(* IEC 61131-3 sources: Codesys/ddyut/src, 26 files *)

(* ---- E_PumpType.st ---- *)
(* ============================================================ *)
(* E_PumpType — тип преобразователя частоты ELHART             *)
(* ============================================================ *)
(* === ИЗМЕНЕНО === MINI удалён (в проектах его не было — была   *)
(* ошибка типа). Теперь два типа: PUMP (EMD-PUMP) и VL           *)
(* (EMD-VL/VH, векторный). Обработка обоих — в FB_Pump.          *)
(*                                                              *)
(* Тип каждого ПЧ задаётся в массиве GVL.ePumpType[1..cPumpCount] *)
(* (RETAIN). Автоопределение PUMP/VL по сигнатурному регистру —   *)
(* см. комментарий в PRG_Pumps (пока задаётся вручную).          *)
(* ============================================================ *)
TYPE E_PumpType :
(
    PUMP := 0,   // EMD-PUMP (F-коды, задание частоты в Гц ×100 → 0x2001)
    VL   := 1    // EMD-VL/VH (P-группы, задание в % → 0x1000, статус 0x3000)
);
END_TYPE

(* ---- GVL.st ---- *)
(* ============================================================ *)
(* GVL — Глобальные переменные проекта ДДЮТ                     *)
(* (на основе Fontan_V1 / Саки Пруд)                            *)
(*                                                              *)
(* ШИНА Modbus RTU / RS-485:                                   *)
(*   COM1 (Modbus_COM), 9600/8/N/1:                            *)
(*     Адрес 1  — МВ110-16Д   (16 дискретных входов DI1..DI11) *)
(*     Адрес 2  — МУ110-16Р   (16 дискретных выходов DO1..DO16)*)
(*     Аналогового модуля МВ110-8А на ДДЮТ НЕТ.                *)
(*   COM2 (Modbus_COM_2):                                       *)
(*     Адрес 41 — ELHART EMD-PUMP 1 (насос фонтана, индекс 1)  *)
(*     Адрес 42 — ELHART EMD-PUMP 2 (насос фонтана, индекс 2)  *)
(*   === ДДЮТ:ИЗМЕНЕНО === Насосы COM2 — это насосы фонтана    *)
(*   (клапаны/форсунки), НЕ фильтрационные, как было в Саки.    *)
(*   Признак работы фильтрации приходит отдельно на DI5.        *)
(* ============================================================ *)

(* ============================================================ *)
(* КОНСТАНТЫ СИСТЕМЫ                                            *)
(* ============================================================ *)
VAR_GLOBAL CONSTANT
    cPumpCount   : INT  := 2;        // количество насосов (2 × EMD-PUMP)
    cDI_Count    : INT  := 16;       // дискретных входов МВ110
    cDO_Count    : INT  := 16;       // дискретных выходов МУ110
    cMaxFreq     : REAL := 50.0;     // максимальная частота, Гц
    cMinFreq     : REAL := 0.0;      // минимальная частота, Гц
    cMinTime     : REAL := 0.1;      // мин. время разгона/торможения, с
    cMaxTime     : REAL := 6000.0;   // макс. время разгона/торможения, с
    cMaxCurrent  : REAL := 999.9;    // потолок номинального тока, А
    cMaxVoltage  : REAL := 500.0;    // потолок номинального напряжения, В
    cMaxOverheat : INT  := 150;      // потолок уровня перегрева, °C
    cMinOverheat : INT  := 40;       // минимум уровня перегрева, °C
END_VAR

(* ============================================================ *)
(* RETAIN-переменные (хранятся при отключении питания)         *)
(* ============================================================ *)
VAR_GLOBAL RETAIN
    (* Тип каждого ПЧ. Оба насоса — EMD-PUMP.                   *)
    (* ВНИМАНИЕ: изменение требует Reset cold контроллера.      *)
    ePumpType : ARRAY[1..cPumpCount] OF E_PumpType :=
        [E_PumpType.PUMP, E_PumpType.PUMP];

    (* === ДДЮТ:ИЗМЕНЕНО (round 7, ФИНАЛЬНАЯ СХЕМА) — ЖУРНАЛ ПЧ === *)
    (* Та же схема сдвига, что у журнала фонтана (см. подробный комментарий  *)
    (* в GVL_Fountain.st) — позиция 1 всегда самая свежая запись, при новой  *)
    (* записи всё сдвигается на 1 вниз, самая старая (позиция 30) выпадает.  *)
    (* Размер: 30 записей (как настроено), длина ячейки 65 (полное время     *)
    (* ДД.ММ.ГГ ЧЧ:ММ:СС + номер ПЧ + название параметра + два REAL-значения *)
    (* — уже было впритык на 65, оставлен без изменений по твоей настройке,  *)
    (* но следи, не обрезаются ли самые длинные названия типа                *)
    (* "Огр.тока.разг" — если увидишь обрыв текста, увеличь до 80-90).       *)
    aPumpLog       : ARRAY[1..30] OF WSTRING(65);
    iPumpLogCount  : INT;   // сколько записей реально заполнено (0..30)

    (* Флаг "задержка ошибки 0x02C0 уже записана в ПЧ" — RETAIN *)
    xErrDelayWritten : ARRAY[1..cPumpCount] OF BOOL := [cPumpCount(FALSE)];

    (* Флаг "параметр дисплея Fout (регистр 0) уже записан" — RETAIN *)
    xDispParamWritten : ARRAY[1..cPumpCount] OF BOOL := [cPumpCount(FALSE)];
END_VAR

(* ============================================================ *)
(* ГЛОБАЛЬНЫЕ ПЕРЕМЕННЫЕ                                        *)
(* ============================================================ *)
VAR_GLOBAL

    (* ========================================================= *)
    (* БЛОК 1: СОСТОЯНИЕ СИСТЕМЫ                                 *)
    (* ========================================================= *)
    xSystemState     : BOOL := TRUE;
    sSystemStateText : WSTRING(20);
    iErrors          : INT  := 0;
    iWorkCount       : INT  := 0;
    iStopCount       : INT  := 0;
    xAnyAlarm        : BOOL := FALSE;
    iErrorsPumps     : INT  := 0;
    iErrorsModules   : INT  := 0;
    iErrorsFountain  : INT  := 0;

    (* ========================================================= *)
    (* БЛОК 2: НАВИГАЦИЯ И ИНТЕРФЕЙС HMI                         *)
    (* ========================================================= *)
    xMenuOpen      : BOOL := TRUE;
    iCurrentScreen : INT  := 1;
    iSelPump       : INT  := 1;

    (* ========================================================= *)
    (* БЛОК 3: РЕЖИМ ОТЛАДКИ RS-485                              *)
    (* ========================================================= *)
    xDebugModeAll      : BOOL := FALSE;
    xDebugModeAll_Prev : BOOL := FALSE;

    xDebugModePump      : ARRAY[1..cPumpCount] OF BOOL := [cPumpCount(FALSE)];
    xDebugModePump_Prev : ARRAY[1..cPumpCount] OF BOOL := [cPumpCount(FALSE)];

    xApplyParamsAll  : BOOL := FALSE;
    xApplyParamsPump : ARRAY[1..cPumpCount] OF BOOL := [cPumpCount(FALSE)];

    (* ========================================================= *)
    (* ТРИГГЕРЫ ЧТЕНИЯ/ЗАПИСИ (конфигуратор-стиль)               *)
    (* ========================================================= *)
    xReadAllPump  : ARRAY[1..cPumpCount] OF BOOL := [cPumpCount(FALSE)];
    xReadAllAsk   : BOOL := FALSE;

    xWriteAllPump : ARRAY[1..cPumpCount] OF BOOL := [cPumpCount(FALSE)];
    xWriteAllAsk  : BOOL := FALSE;
    xWriteAllConfirm : BOOL := FALSE;

    xWr_AccTime      : ARRAY[1..cPumpCount] OF BOOL := [cPumpCount(FALSE)]; // 0x006B
    xWr_DecTime      : ARRAY[1..cPumpCount] OF BOOL := [cPumpCount(FALSE)]; // 0x006C
    xWr_MaxFreq      : ARRAY[1..cPumpCount] OF BOOL := [cPumpCount(FALSE)]; // 0x0069
    xWr_MinFreq      : ARRAY[1..cPumpCount] OF BOOL := [cPumpCount(FALSE)]; // 0x006A
    xWr_MotorCurrent : ARRAY[1..cPumpCount] OF BOOL := [cPumpCount(FALSE)]; // 0x00D2
    xWr_MotorVoltage : ARRAY[1..cPumpCount] OF BOOL := [cPumpCount(FALSE)]; // 0x00D1
    xWr_OverCurLevel : ARRAY[1..cPumpCount] OF BOOL := [cPumpCount(FALSE)]; // 0x01A7
    xWr_OverCurTime  : ARRAY[1..cPumpCount] OF BOOL := [cPumpCount(FALSE)]; // 0x01A8
    xWr_OverVoltProt : ARRAY[1..cPumpCount] OF BOOL := [cPumpCount(FALSE)]; // 0x019B
    xWr_Overheat     : ARRAY[1..cPumpCount] OF BOOL := [cPumpCount(FALSE)]; // 0x0325
    xWr_OverCurAcc   : ARRAY[1..cPumpCount] OF BOOL := [cPumpCount(FALSE)]; // 0x0199

    xWr_UnlockF800   : ARRAY[1..cPumpCount] OF BOOL := [cPumpCount(FALSE)]; // 0x0320
    xWr_Sources      : ARRAY[1..cPumpCount] OF BOOL := [cPumpCount(FALSE)]; // 0x0065/0x0066

    xWritePending    : ARRAY[1..cPumpCount] OF BOOL := [cPumpCount(FALSE)];
    xWaitStopForWrite : ARRAY[1..cPumpCount] OF BOOL := [cPumpCount(FALSE)];

    (* === ДДЮТ:УДАЛИТЬ ===                                       *)
    (* Раньше использовался для запроса физической остановки      *)
    (* фильтр.насоса через лампы DO6/DO8 перед записью параметров. *)
    (* На ДДЮТ ПЧ COM2 — насосы фонтана, ламп-повторов DI4/DI5     *)
    (* больше нет (DO6/DO8 свободны). Остановка перед записью      *)
    (* параметров идёт командой Modbus (см. PRG_Pumps, источник    *)
    (* RS-485) — эта переменная физически нигде не читается,      *)
    (* оставлена только для истории. Можно удалить совсем.        *)
    xReqStopFiltrForWrite : ARRAY[1..cPumpCount] OF BOOL := [cPumpCount(FALSE)];

    xFactoryResetAll  : BOOL := FALSE;
    xFactoryResetPump : ARRAY[1..cPumpCount] OF BOOL := [cPumpCount(FALSE)];

    wCmdSourceWrite  : ARRAY[1..cPumpCount] OF WORD := [cPumpCount(WORD#1)];
    wFreqSourceWrite : ARRAY[1..cPumpCount] OF WORD := [cPumpCount(WORD#3)];

    (* ========================================================= *)
    (* БЛОК 4: МВ110-16Д — ДИСКРЕТНЫЕ ВХОДЫ                      *)
    (* ========================================================= *)
    wMV110_Inputs : WORD;
    xMV110_Error  : BOOL;
    xDI           : ARRAY[1..cDI_Count] OF BOOL;
    (* === ДДЮТ:ИЗМЕНЕНО === Используются DI1..DI11.             *)
    (* Карта DI — см. PRG_Fountain блок 2.                       *)

    (* ========================================================= *)
    (* БЛОК 5: МУ110-16Р — ДИСКРЕТНЫЕ ВЫХОДЫ                     *)
    (* ========================================================= *)
    (* === ДДЮТ:ИЗМЕНЕНО === Карта DO1..DO16 — см. PRG_Fountain   *)
    (* блок 17. DO1 свет, DO2 авария, DO9 насосы, DO11 добор,     *)
    (* DO13 сухой ход/разрешение (инверсия аварии добора),        *)
    (* DO14 альгицид, DO15 биопаг, DO16 pH. Остальные свободны.   *)
    xDO                : ARRAY[1..cDO_Count] OF BOOL := [cDO_Count(FALSE)];

    wMU110_Outputs     : WORD := 0;
    wMU110_OutputsRead : WORD;
    xMU110_Error       : BOOL;

    wMU110_SafeOutputs : WORD := 0;
    xMU110_WriteSafe   : BOOL := FALSE;

    (* ========================================================= *)
    (* БЛОК 6: НАСОСЫ — ЭКЗЕМПЛЯРЫ ФУНКЦИОНАЛЬНЫХ БЛОКОВ         *)
    (* ========================================================= *)
    Pump : ARRAY[1..cPumpCount] OF FB_Pump;

    (* ========================================================= *)
    (* БЛОК 7: НАСОСЫ — ЗАДАНИЕ ОПЕРАТОРА (_Set)                 *)
    (* ========================================================= *)
    xPumpRunCmd : ARRAY[1..cPumpCount] OF BOOL := [cPumpCount(FALSE)];

    rPumpFreqSetHz          : ARRAY[1..cPumpCount] OF REAL := [cPumpCount(40.0)];
    rPumpAccTime_Set        : ARRAY[1..cPumpCount] OF REAL := [10.0, 10.0];
    rPumpDecTime_Set        : ARRAY[1..cPumpCount] OF REAL := [10.0, 10.0];
    rPumpMaxFreq_Set        : ARRAY[1..cPumpCount] OF REAL := [cPumpCount(40.0)];
    rPumpMinFreq_Set        : ARRAY[1..cPumpCount] OF REAL := [cPumpCount(0.0)];
    rPumpMotorRatedCurrent_Set : ARRAY[1..cPumpCount] OF REAL := [cPumpCount(14.9)];
    rPumpMotorRatedVoltage_Set : ARRAY[1..cPumpCount] OF REAL := [cPumpCount(380.0)];
    rPumpOverCurrentLevel_A_Set : ARRAY[1..cPumpCount] OF REAL := [cPumpCount(26.1)];
    rPumpOverCurrentTime_Set    : ARRAY[1..cPumpCount] OF REAL := [cPumpCount(5.0)];
    xPumpOverVoltProtect_Set    : ARRAY[1..cPumpCount] OF BOOL := [cPumpCount(TRUE)];
    iPumpOverheatLevel_Set      : ARRAY[1..cPumpCount] OF INT  := [cPumpCount(95)];
    iPumpOverCurAcc_Set         : ARRAY[1..cPumpCount] OF INT  := [cPumpCount(150)];

    (* ========================================================= *)
    (* БЛОК 7а: ОТЛАДКА — групповые команды и флаги окон        *)
    (* ========================================================= *)
    xDbgRunAll  : BOOL;
    xDbgStopAll : BOOL;

    xAskApply   : BOOL := FALSE;
    xAskFactory : BOOL := FALSE;
	xAskDialogStopPch : BOOL := FALSE;

    (* ========================================================= *)
    (* БЛОК 8: НАСОСЫ — ДАННЫЕ ДЛЯ ОТОБРАЖЕНИЯ НА HMI            *)
    (* ========================================================= *)
    xPumpWork      : ARRAY[1..cPumpCount] OF BOOL;
    xPumpStop      : ARRAY[1..cPumpCount] OF BOOL;
    xPumpAlarm     : ARRAY[1..cPumpCount] OF BOOL;
    xPumpReverse   : ARRAY[1..cPumpCount] OF BOOL;
    xPumpCommError : ARRAY[1..cPumpCount] OF BOOL;
    xPumpCommRaw   : ARRAY[1..cPumpCount] OF BOOL;
    tonPumpCommFilter : ARRAY[1..cPumpCount] OF TON;

    sPumpState         : ARRAY[1..cPumpCount] OF WSTRING(50);
    sPumpFaultText     : ARRAY[1..cPumpCount] OF WSTRING(100);
    sPumpTypeText      : ARRAY[1..cPumpCount] OF WSTRING(20);
    sPumpFaultLastText : ARRAY[1..cPumpCount] OF WSTRING(100);
    sPumpFault2Text    : ARRAY[1..cPumpCount] OF WSTRING(100);
    sPumpFault3Text    : ARRAY[1..cPumpCount] OF WSTRING(100);
    sPumpFault4Text    : ARRAY[1..cPumpCount] OF WSTRING(100);

    rPumpFreqSetActHz : ARRAY[1..cPumpCount] OF REAL;
    rPumpFreqActHz    : ARRAY[1..cPumpCount] OF REAL;
    rPumpCurrentActA  : ARRAY[1..cPumpCount] OF REAL;
    rPumpSpeedActRpm  : ARRAY[1..cPumpCount] OF REAL;
    rPumpDcVoltageV   : ARRAY[1..cPumpCount] OF REAL;
    iPumpTemperatureC : ARRAY[1..cPumpCount] OF INT;
    rPumpVoltageActV  : ARRAY[1..cPumpCount] OF REAL;
    rPumpRuntimeHours : ARRAY[1..cPumpCount] OF REAL;

    dwPumpLampColor : ARRAY[1..cPumpCount] OF DWORD;

    rPumpAccTime_Disp            : ARRAY[1..cPumpCount] OF REAL;
    rPumpDecTime_Disp            : ARRAY[1..cPumpCount] OF REAL;
    rPumpMaxFreq_Disp            : ARRAY[1..cPumpCount] OF REAL;
    rPumpMinFreq_Disp            : ARRAY[1..cPumpCount] OF REAL;
    rPumpMotorRatedCurrent_Disp  : ARRAY[1..cPumpCount] OF REAL;
    rPumpMotorRatedVoltage_Disp  : ARRAY[1..cPumpCount] OF REAL;
    rPumpOverCurrentLevel_A_Disp : ARRAY[1..cPumpCount] OF REAL;
    rPumpOverCurrentTime_Disp    : ARRAY[1..cPumpCount] OF REAL;
    xPumpOverVoltProtect_Disp    : ARRAY[1..cPumpCount] OF BOOL;
    sPumpOverVoltProtect : ARRAY[1..cPumpCount] OF WSTRING(20);
    iPumpOverCurrentLevel_pct_Disp : ARRAY[1..cPumpCount] OF INT;
    iPumpOverheatLevel_Disp      : ARRAY[1..cPumpCount] OF INT;
    iPumpOverCurAcc_Disp         : ARRAY[1..cPumpCount] OF INT;

    (* ========================================================= *)
    (* БЛОК 9: НАСОСЫ — ЗАПИСЬ В ПЧ (Modbus WRITE)               *)
    (* ========================================================= *)
    wPumpCmd  : ARRAY[1..cPumpCount] OF WORD;
    wPumpFreq : ARRAY[1..cPumpCount] OF WORD;

    wPumpAccTimeWrite           : ARRAY[1..cPumpCount] OF WORD;
    wPumpDecTimeWrite           : ARRAY[1..cPumpCount] OF WORD;
    wPumpMaxFreqWrite           : ARRAY[1..cPumpCount] OF WORD;
    wPumpMinFreqWrite           : ARRAY[1..cPumpCount] OF WORD;
    wPumpMotorRatedCurrentWrite : ARRAY[1..cPumpCount] OF WORD;
    wPumpMotorRatedVoltageWrite : ARRAY[1..cPumpCount] OF WORD;
    wPumpOverCurrentLevelWrite  : ARRAY[1..cPumpCount] OF WORD;
    wPumpOverCurrentTimeWrite   : ARRAY[1..cPumpCount] OF WORD;
    wPumpOverVoltProtectWrite   : ARRAY[1..cPumpCount] OF WORD;
    wPumpOverheatLevelWrite     : ARRAY[1..cPumpCount] OF WORD;
    wPumpOverCurAccWrite        : ARRAY[1..cPumpCount] OF WORD;

    wPumpDispParamWrite : ARRAY[1..cPumpCount] OF WORD := [cPumpCount(WORD#1)];

    wPumpRS_ErrDelayWrite : ARRAY[1..cPumpCount] OF WORD := [cPumpCount(WORD#5)];
    xWr_ErrDelayInit      : ARRAY[1..cPumpCount] OF BOOL := [cPumpCount(FALSE)];

    wPumpExtSettingsUnlockWrite : ARRAY[1..cPumpCount] OF WORD;
    wPumpFactoryResetWrite      : ARRAY[1..cPumpCount] OF WORD := [cPumpCount(WORD#0)];

    (* ========================================================= *)
    (* БЛОК 10: НАСОСЫ — ЧТЕНИЕ ИЗ ПЧ (Modbus READ)             *)
    (* ========================================================= *)
    wPumpFreqSetRead     : ARRAY[1..cPumpCount] OF WORD;
    wPumpFreqActual      : ARRAY[1..cPumpCount] OF WORD;
    wPumpCurrentActual   : ARRAY[1..cPumpCount] OF WORD;
    wPumpSpeedActual     : ARRAY[1..cPumpCount] OF WORD;
    wPumpDcVoltage       : ARRAY[1..cPumpCount] OF WORD;
    wPumpTemperature     : ARRAY[1..cPumpCount] OF WORD;
    wPumpPidFeedback     : ARRAY[1..cPumpCount] OF WORD;
    wPumpRuntimeHoursRaw : ARRAY[1..cPumpCount] OF WORD;
    wPumpVoltageActual   : ARRAY[1..cPumpCount] OF WORD;

    wPumpFaultLast : ARRAY[1..cPumpCount] OF WORD;
    wPumpFault2    : ARRAY[1..cPumpCount] OF WORD;
    wPumpFault3    : ARRAY[1..cPumpCount] OF WORD;
    wPumpFault4    : ARRAY[1..cPumpCount] OF WORD;

    wPumpFaultReg : ARRAY[1..cPumpCount] OF WORD;
    wPumpStatus   : ARRAY[1..cPumpCount] OF WORD;
    wPumpStopState    : ARRAY[1..cPumpCount] OF WORD;
    xPumpFullyStopped : ARRAY[1..cPumpCount] OF BOOL;

    wPumpFreqPresetRead  : ARRAY[1..cPumpCount] OF WORD;
    rPumpFreqPresetHz : ARRAY[1..cPumpCount] OF REAL;
    wPumpFreqSourceRead  : ARRAY[1..cPumpCount] OF WORD;
    wPumpCmdSourceRead   : ARRAY[1..cPumpCount] OF WORD;
    wPumpStopKeyLockRead : ARRAY[1..cPumpCount] OF WORD;
    wPumpReverseLockRead : ARRAY[1..cPumpCount] OF WORD;
    wPumpMaxFreqRead     : ARRAY[1..cPumpCount] OF WORD;
    wPumpMinFreqRead     : ARRAY[1..cPumpCount] OF WORD;
    wPumpAccTimeRaw      : ARRAY[1..cPumpCount] OF WORD;
    wPumpDecTimeRaw      : ARRAY[1..cPumpCount] OF WORD;

    wPumpStartMethodRead        : ARRAY[1..cPumpCount] OF WORD;
    wPumpStopMethodRead         : ARRAY[1..cPumpCount] OF WORD;
    wPumpStartFreqRead          : ARRAY[1..cPumpCount] OF WORD;
    wPumpStopFreqRead           : ARRAY[1..cPumpCount] OF WORD;
    wPumpMotorRatedVoltageRead  : ARRAY[1..cPumpCount] OF WORD;
    wPumpMotorRatedCurrentRead  : ARRAY[1..cPumpCount] OF WORD;
    wPumpMotorNoLoadCurrentRead : ARRAY[1..cPumpCount] OF WORD;
    wPumpMotorRatedSpeedRead    : ARRAY[1..cPumpCount] OF WORD;

    wPumpFIV_MinRead    : ARRAY[1..cPumpCount] OF WORD;
    wPumpFIV_MaxRead    : ARRAY[1..cPumpCount] OF WORD;
    wPumpFIV_FilterRead : ARRAY[1..cPumpCount] OF WORD;
    wPumpFIC_MinRead    : ARRAY[1..cPumpCount] OF WORD;
    wPumpFIC_MaxRead    : ARRAY[1..cPumpCount] OF WORD;

    wPumpFOV_MinRead : ARRAY[1..cPumpCount] OF WORD;
    wPumpFOV_MaxRead : ARRAY[1..cPumpCount] OF WORD;
    wPumpFOC_MinRead : ARRAY[1..cPumpCount] OF WORD;
    wPumpFOC_MaxRead : ARRAY[1..cPumpCount] OF WORD;

    wPumpAI_MinFreqRead  : ARRAY[1..cPumpCount] OF WORD;
    wPumpAI_MinDirRead   : ARRAY[1..cPumpCount] OF WORD;
    wPumpAI_MaxFreqRead  : ARRAY[1..cPumpCount] OF WORD;
    wPumpAI_MaxDirRead   : ARRAY[1..cPumpCount] OF WORD;
    wPumpAI_ReverseEnRead: ARRAY[1..cPumpCount] OF WORD;

    wPumpDI_FWD_Read : ARRAY[1..cPumpCount] OF WORD;
    wPumpDI_REV_Read : ARRAY[1..cPumpCount] OF WORD;
    wPumpDI_S1_Read  : ARRAY[1..cPumpCount] OF WORD;
    wPumpDI_S2_Read  : ARRAY[1..cPumpCount] OF WORD;
    wPumpDI_S3_Read  : ARRAY[1..cPumpCount] OF WORD;
    wPumpDI_S4_Read  : ARRAY[1..cPumpCount] OF WORD;
    wPumpDI_S5_Read  : ARRAY[1..cPumpCount] OF WORD;
    wPumpDI_S6_Read  : ARRAY[1..cPumpCount] OF WORD;

    wPumpDO_M01_Read   : ARRAY[1..cPumpCount] OF WORD;
    wPumpDO_M02_Read   : ARRAY[1..cPumpCount] OF WORD;
    wPumpDO_Relay_Read : ARRAY[1..cPumpCount] OF WORD;

    wPumpOverCurAccRead       : ARRAY[1..cPumpCount] OF WORD;
    wPumpOverCurSteadyRead    : ARRAY[1..cPumpCount] OF WORD;
    wPumpOverVoltProtectRead  : ARRAY[1..cPumpCount] OF WORD;
    wPumpOverCurReactionRead  : ARRAY[1..cPumpCount] OF WORD;
    wPumpOverCurrentLevelRead : ARRAY[1..cPumpCount] OF WORD;
    wPumpOverCurrentTimeRead  : ARRAY[1..cPumpCount] OF WORD;
    wPumpOverheatLevelRead    : ARRAY[1..cPumpCount] OF WORD;

    wPumpRS_BaudRead      : ARRAY[1..cPumpCount] OF WORD;
    wPumpRS_FormatRead    : ARRAY[1..cPumpCount] OF WORD;
    wPumpRS_AddrRead      : ARRAY[1..cPumpCount] OF WORD;
    wPumpRS_ErrActionRead : ARRAY[1..cPumpCount] OF WORD;
    wPumpRS_ErrDelayRead  : ARRAY[1..cPumpCount] OF WORD;

    (* ========================================================= *)
    (* БЛОК 11: VISU DEBUG — ВЫБОР НАСОСА И ДИАЛОГИ              *)
    (* ========================================================= *)
    iDebugMode         : INT;
    iDebugPumpSelected : INT := 1;
    xDlgConfirmApply   : BOOL;
    xDlgConfirmFactory : BOOL;

(* ========================================================= *)
(* БЛОК 12: ЖУРНАЛ ИЗМЕНЕНИЙ ПАРАМЕТРОВ ПЧ *)
(* ========================================================= *)
xLogClear : BOOL := FALSE;
xAskClearLog : BOOL := FALSE;

rLog_AccTime_Prev : ARRAY[1..cPumpCount] OF REAL;
rLog_DecTime_Prev : ARRAY[1..cPumpCount] OF REAL;
rLog_MaxFreq_Prev : ARRAY[1..cPumpCount] OF REAL;
rLog_MinFreq_Prev : ARRAY[1..cPumpCount] OF REAL;
rLog_MotorCur_Prev : ARRAY[1..cPumpCount] OF REAL;
rLog_MotorVolt_Prev : ARRAY[1..cPumpCount] OF REAL;
rLog_OCLevel_Prev : ARRAY[1..cPumpCount] OF REAL;
rLog_OCTime_Prev : ARRAY[1..cPumpCount] OF REAL;
xLog_OVProt_Prev : ARRAY[1..cPumpCount] OF BOOL;
iLog_Overheat_Prev : ARRAY[1..cPumpCount] OF INT;
iLog_OCAcc_Prev : ARRAY[1..cPumpCount] OF INT;
xLog_Initialized : ARRAY[1..cPumpCount] OF BOOL := [cPumpCount(FALSE)];
rtrigReadAll_Prev : ARRAY[1..cPumpCount] OF BOOL := [cPumpCount(FALSE)];

xWr_DispParam : ARRAY[1..cPumpCount] OF BOOL := [cPumpCount(FALSE)];
END_VAR

(* ---- GVL_Fountain.st ---- *)
(* ============================================================ *)
(* GVL_Fountain — переменные автоматики фонтана ДДЮТ            *)
(* (на основе Fontan_V1 / Саки Пруд)                            *)
(*                                                              *)
(* === ГЛАВНЫЕ ОТЛИЧИЯ ОТ САКИ ===                              *)
(*  - Уровень чаши: ДВА дискретных входа (DI7 нижний, DI8       *)
(*    верхний) вместо аналогового 4-20мА. Нет ямы слива.        *)
(*  - Сухой ход — отдельный вход DI6, не расчёт по см.          *)
(*  - Фильтрация: контактор фильтр.насоса на DI5 отдельно от    *)
(*    насосов COM2 (те теперь качают фонтан, не фильтруют).     *)
(*  - Нет ПР200 и резерва полива СПК (файлы сохранены, не       *)
(*    вызываются — легко вернуть).                              *)
(*  - Расчёт заката — новый (NOAA, FB_SunsetRelay), не завязан   *)
(*    ни на один DI.                                            *)
(*                                                              *)
(* КАРТА ВЫХОДОВ DO (МУ110-16Р, COM1, адрес 2):                 *)
(*   DO1  — СВЕТ                                                *)
(*   DO2  — ЛАМПА АВАРИИ (мигает)                                *)
(*   DO3..DO8, DO10, DO12 — свободны (FALSE)                    *)
(*   DO9  — НАСОСЫ ФОНТАНА                                      *)
(*   DO11 — КЛАПАН ДОБОРА (заслонка)                            *)
(*   DO13 — "сухой ход/разрешение": 1=норма, 0=авария добора    *)
(*          (после исчерпания попыток), см. PRG_Fountain блок 7 *)
(*   DO14 — АЛЬГИЦИД                                             *)
(*   DO15 — БИОПАГ / ОБЕЗЗАРАЖИВАТЕЛЬ                            *)
(*   DO16 — pH                                                  *)
(*                                                              *)
(* КАРТА ВХОДОВ DI (МВ110-16Д, COM1, адрес 1):                  *)
(*   DI1  — ПЧ1 насос фонтана (работа)                          *)
(*   DI2  — ПЧ2 насос фонтана (работа)                          *)
(*   DI3  — разрешение работы частотников                       *)
(*   DI4  — контактор УФ (мониторинг, выхода на УФ нет)         *)
(*   DI5  — контактор фильтр.насоса (наработка НФ)               *)
(*   DI6  — реле СУХОГО ХОДА (1 = вода есть)                    *)
(*   DI7  — УРОВЕНЬ 1 нижний  (0 = нужен добор)                 *)
(*   DI8  — УРОВЕНЬ 2 верхний (1 = стоп добора)                 *)
(*   DI9  — подтверждение работы pH                             *)
(*   DI10 — подтверждение работы биопаг                         *)
(*   DI11 — подтверждение работы альгицид                       *)
(*   DI12..DI16 — свободны                                       *)
(* ============================================================ *)

VAR_GLOBAL CONSTANT
    (* === ДДЮТ:УДАЛИТЬ — шкала уровня чаши по AI1 не нужна === *)
    (* Уровень чаши теперь дискретный (DI7/DI8), нет 4-20мА.     *)
    (*
    cWaterRawMin : REAL := 4.0;
    cWaterRawMax : REAL := 20.0;
    cWaterCmMin  : REAL := 0.0;
    cWaterCmMax  : REAL := 100.0;
    *)

    (* === ДДЮТ: ОСТАВЛЕНО АКТИВНЫМ === Используется только      *)
    (* файлом PRG_PolivSPK.st (сохранён, не вызывается на ДДЮТ,  *)
    (* т.к. нет ямы слива). Оставлено, чтобы файл не переставал   *)
    (* компилироваться. Если PRG_PolivSPK.st будет физически      *)
    (* удалён из проекта — эти константы тоже можно убрать.       *)
    cSlivRawMin : REAL := 4.0;
    cSlivRawMax : REAL := 20.0;
    cSlivCmMin  : REAL := 0.0;
    cSlivCmMax  : REAL := 100.0;
END_VAR

VAR_GLOBAL RETAIN
    (* === ДДЮТ:ИЗМЕНЕНО (round 7, ФИНАЛЬНАЯ СХЕМА) — ЖУРНАЛ ИЗМЕНЕНИЙ       *)
    (* ПАРАМЕТРОВ ФОНТАНА ===                                                 *)
    (* Причина, почему это массив, а не одна строка — см. round 6: WCONCAT в *)
    (* CODESYS официально ограничен 255 символами возврата, независимо от     *)
    (* объявленного размера WSTRING (https://content.helpme-codesys.com/en/  *)
    (* CODESYS String Libraries/_strlib_start_page.html).                    *)
    (* === ДДЮТ:ИЗМЕНЕНО (round 7) === СХЕМА СДВИГА (новое): позиция 1 —      *)
    (* ВСЕГДА самая последняя запись. При каждой новой записи всё, что было,  *)
    (* сдвигается на 1 позицию вниз (2→3, 1→2), новая запись садится на       *)
    (* позицию 1. Когда достигнут предел (60) — самая старая запись           *)
    (* (позиция 60) при сдвиге просто "выпадает" из массива. Это устраняет    *)
    (* необходимость в НА ЭКРАНЕ вычисляемых индексах вида                    *)
    (* "aFountainLog[iFountainLogCount-k]" — ИМЕННО такие вычисляемые         *)
    (* индексы, судя по всему, и давали "путаницу переменных" (при           *)
    (* iFountainLogCount меньше, чем число видимых на экране строк, индекс    *)
    (* уходил в 0 или отрицательное число — обращение к несуществующему       *)
    (* элементу массива в CODESYS не ошибка компиляции, а чтение "что         *)
    (* попало" из соседней памяти). Теперь на экране — ВСЕГДА статичные       *)
    (* константы 1, 2, 3... — вне диапазона массива уйти невозможно.          *)
    (* Размер: 60 записей, длина ячейки 60 символов (по прямому запросу).    *)
    (* ⚠️ С полными названиями + единицы измерения у обоих значений + пробелы*)
    (* вокруг стрелки — для записей с REAL (доза/расход, REAL_TO_WSTRING     *)
    (* может дать много знаков после запятой) возможна обрезка в конце       *)
    (* строки при длинных значениях. Если увидишь обрыв текста — увеличивай.*)
    aFountainLog       : ARRAY[1..60] OF WSTRING(60);
    iFountainLogCount  : INT;   // сколько записей реально заполнено (0..60)

    (* === ДДЮТ:НОВОЕ === Единый пароль для очистки ОБОИХ журналов        *)
    (* (ПЧ и фонтана) — числовой, проверяется в ST-коде через встроенный   *)
    (* элемент OwenVisu LoginOnlyPassWithKeysOwen. RETAIN — не теряется    *)
    (* при пропадании питания. Поменяй значение под себя (это заводское    *)
    (* значение-пример, не оставляй в эксплуатации).                       *)
    iAdminPassCorrect : INT := 1234;

    (* ===== ГЛАВНЫЕ ТУМБЛЕРЫ С ЭКРАНА ====================== *)
    xVseSist : BOOL := TRUE;
    (* === ДДЮТ:ИЗМЕНЕНО (единый селектор режимов) ===          *)
    (* Вместо двух раздельных элементов (тумблер разрешения +    *)
    (* отдельная кнопка ручного пуска) — один 3-позиционный      *)
    (* выбор на экране, который сам раскладывается на пару       *)
    (* (Enable, ManualForce). Раскладка — в PRG_Fountain.st,      *)
    (* блок 2а. Значения:                                        *)
    (*   0 = Ручной пуск (принудительно вкл, минуя автоматику)   *)
    (*   1 = Выкл (запрет) — значение по умолчанию для ЛЮБОГО     *)
    (*       некорректного индекса тоже трактуется как "выкл"    *)
    (*   2 = Авто (штатная логика с учётом всех условий)         *)
    iPumpSelect : INT := 2;   // насосы фонтана: 0=ручной,1=выкл,2=авто
    xNfEnable : BOOL := TRUE;

    (* ===== === ДДЮТ:УДАЛИТЬ — УСТАВКИ УРОВНЯ В СМ (AI1) ===== *)
    (* Уровень теперь дискретный, пороги в см не нужны.          *)
    (*
    rLevelOverflow   : REAL := 94.0;
    rLevelNorm       : REAL := 92.5;
    rLevelRefill     : REAL := 91.5;
    rLevelEmergency1 : REAL := 88.0;
    rLevelEmergency2 : REAL := 60.0;
    sLevelOverflow : WSTRING := "Уровень Перелив";
    sLevelNorm : WSTRING := "Уровень Норма";
    sLevelRefill : WSTRING := "Уровень Подпитка";
    sLevelEmergency1 : WSTRING := "Уровень Аварийный 1";
    sLevelEmergency2 : WSTRING := "Уровень Перелив Аварийный 2";
    *)

    (* ===== === ДДЮТ:ИЗМЕНЕНО — УРОВЕНЬ, КОНФИГУРИРУЕМЫЙ 2 ИЛИ 3   *)
    (* ДАТЧИКА (с экрана, кнопками/тумблером) ================= *)
    (* iLevelSensorCountPending = 2: датчики Уровень1 (DI7) и Уровень2*)
    (* (DI8).                                                        *)
    (*   Уровень1=0 (подтверждено) → СУХОЙ ХОД (запрет всего).     *)
    (*   Уровень1=1 И Уровень2=0 (подтверждено) → СТАРТ добора.    *)
    (*   Уровень2=1 (подтверждено) → "хватит", ПОСЛЕ доп.задержки  *)
    (*   iRefillOffDelayMin/Sec — СТОП добора.                     *)
    (* iLevelSensorCountPending = 3: датчики Уровень1 (DI7), Уровень2*)
    (* (DI8), Уровень3 (DI12).                                      *)
    (*   Уровень1=0 (подтверждено) → СУХОЙ ХОД (запрет всего) —     *)
    (*   РОЛЬ ТА ЖЕ, что и в режиме на 2 датчика.                   *)
    (*   Уровень2=0 (подтверждено) → СТАРТ добора (та же роль,      *)
    (*   что у Уровня2 в режиме на 2 датчика).                      *)
    (*   Уровень3=1 (подтверждено) → "хватит", ПОСЛЕ доп.задержки   *)
    (*   — СТОП добора (роль, которую в 2-датчиковом режиме играет  *)
    (*   сам Уровень2).                                             *)
    (* Итог: Уровень1 везде = сухой ход. Уровень2 везде = старт      *)
    (* добора. Разница только в том, ОТКУДА берётся сигнал "хватит":*)
    (* в 2-датчиковом режиме — снова Уровень2 (=1), в 3-датчиковом  *)
    (* — отдельный Уровень3.                                        *)
    (* === ДДЮТ:ИЗМЕНЕНО === Раньше было две переменные (Pending +   *)
    (* подтверждённая, с диалогом PIN-подтверждения в коде). Убрано  *)
    (* по твоей просьбе — защита от случайной записи теперь делается *)
    (* штатными средствами CODESYS (права доступа/пароль на элемент  *)
    (* визуализации при записи переменной), отдельная ST-логика для  *)
    (* этого не нужна. Осталась ОДНА переменная, пишется с экрана     *)
    (* напрямую, используется везде по коду как есть.                *)
    iLevelSensorCountPending : INT := 2;   // 2 или 3, пишется с экрана напрямую

    (* === ДДЮТ:УДАЛИТЬ === "потолок времени" был временной заменой   *)
    (* системы попыток (см. tRefillDurHours/tBetweenRefillHours/       *)
    (* iRefillAttemptsMax выше) — вернул как было в Саки, эта одиночная*)
    (* уставка больше не нужна.                                        *)
    (*
    iRefillMaxDurationMin : INT := 90;
    *)

    (* Гистерезис (антидребезг) КАЖДОГО датчика — свой, все         *)
    (* редактируются с экрана. По умолчанию 20 сек.                 *)
    tLevel1DebounceSec : INT := 20;  // Уровень1 (сухой ход)
    tLevel2DebounceSec : INT := 20;  // Уровень2 (старт добора; и стоп в режиме 2 датчика)
    tLevel3DebounceSec : INT := 20;  // Уровень3 (стоп добора, ТОЛЬКО режим 3 датчика)

    (* Доп. задержка ВЫКЛЮЧЕНИЯ добора после того, как "хватит"      *)
    (* подтверждено гистерезисом — чтобы не дёргать клапан сразу.   *)
    (* Задаётся в минутах+секундах с экрана. По умолчанию 2 мин 0с. *)
    (* Если поставить 0:00 — выключение происходит сразу (без доп.  *)
    (* выдержки), работает в обоих режимах (2 и 3 датчика) одинаково.*)
    iRefillOffDelayMin : INT := 2;
    iRefillOffDelaySec : INT := 0;

    (* === ДДЮТ:УДАЛИТЬ — ПАРАМЕТРЫ ЗАСЛОНКИ ПО КОНЦЕВИКАМ =========*)
    (* Не применимы — на ДДЮТ у заслонки нет концевиков/реле         *)
    (* направления, только команда клапана.                         *)
    (*
    tDamperTimeoutSec   : INT := 60;
    tOverflowDelaySec   : INT := 60;
    tLevelBlockDelaySec : INT := 10;
    tDamperConfirmSec : INT := 20;
    *)

    (* Смещение часового пояса от UTC, сек. Крым/МСК = +3ч=10800.*)
    iTimeZoneOffsetSec : INT := 10800;
    iUvNfMinRunMin : INT := 20;   // мин. непрерывной работы НФ для включения УФ, мин (перепроверить)

    (* === ДДЮТ:ВОЗВРАЩЕНО — СИСТЕМА ПОПЫТОК ДОБОРА === *)
    (* Была помечена "устарела" и заменена простым потолком времени  *)
    (* (xRefillMaxDurationAlarm) — но это было неверно: одна неудачная *)
    (* попытка (например, временно нет воды в городском водопроводе) *)
    (* не должна сразу давать аварию. Возвращена логика из Саки:      *)
    (* пробуем добраться tRefillDurHours; если не вышло — пауза       *)
    (* tBetweenRefillHours, новая попытка; после iRefillAttemptsMax   *)
    (* неудачных попыток подряд — авария, до ручного сброса.          *)
    (* xRefillMaxDurationAlarm/iRefillMaxDurationMin — УДАЛЕНЫ,       *)
    (* эта система их полностью заменяет.                             *)
    tRefillDurHours     : INT := 2;   // время на одну попытку добора, часы
    tBetweenRefillHours : INT := 12;  // пауза между неудачными попытками, часы
    iRefillAttemptsMax  : INT := 5;   // макс. число неудачных попыток подряд

    (* === ДДЮТ:УДАЛИТЬ — пороги сливного бака (нет ямы слива) === *)
    (*
    rSlivPolivOnCm : REAL := 5.0;
    rSlivDoborOnCm : REAL := 20.0;
    rSlivNormaPolivCm : REAL := 30.0;
    *)

    (* ===== ДОЗАЦИЯ pH — ТОЛЬКО РАЗРЕШЕНИЕ (без таймера) ==== *)
    (* === ДДЮТ:ИЗМЕНЕНО (единый селектор) — см. пояснение у   *)
    (* iPumpSelect выше. Раскладка в PRG_Fountain.st блок 2а.   *)
    iPhSelect : INT := 2;   // pH: 0=ручной,1=выкл,2=авто

    (* ===== ДОЗАЦИЯ АЛЬГИЦИД — === ДДЮТ:ИЗМЕНЕНО (round 3), реальные значения === *)
    iAlgSelect        : INT := 2;   // альгицид: 0=ручной,1=выкл,2=авто
    rAlgDoseMlPerDay  : REAL := 66.0;     // суточная доза, мл (ДДЮТ)
    rAlgFlowMlPerHour : REAL := 1125.0;   // расход насоса, мл/ч (ДДЮТ)

    (* ===== ДОЗАЦИЯ БИОПАГА — === ДДЮТ:ИЗМЕНЕНО (round 3), реальные значения === *)
    (* ВНИМАНИЕ — МОЯ ИНТЕРПРЕТАЦИЯ ЧИСЕЛ, ПРОВЕРЬ:                *)
    (* Ты написал расход "1.125 и 1.154" без единиц. Для альгицида *)
    (* уже подтверждено 1125 мл/ч (совпадает с "1.125" при чтении   *)
    (* точки как разделителя тысяч). По той же логике "1.154"       *)
    (* прочитано как 1154 мл/ч (а не буквально 1.154 мл/ч — при     *)
    (* таком мизерном расходе доза 33 мл выдавалась бы ~29 часов,    *)
    (* что маловероятно). Если я неправильно понял и расход         *)
    (* биопага ДЕЙСТВИТЕЛЬНО 1.154 мл/ч (не 1154) — поменяй ниже.   *)
    iBioSelect        : INT := 2;   // биопаг: 0=ручной,1=выкл,2=авто
    rBioDoseMlPerDay  : REAL := 33.0;     // суточная доза, мл (ДДЮТ)
    rBioFlowMlPerHour : REAL := 1154.0;   // расход насоса, мл/ч (ДДЮТ) — СВЕРИТЬ, см. выше

    (* ===== ОКНО ИСПРАВНОСТИ ФИЛЬТРАЦИИ ==================== *)
    iFilterMinRunMin   : INT := 30;    // порог наработки НФ, мин (перепроверить)
    iFilterWindowHours : INT := 12;    // (устар., не используется)
    iNfHealthyWindowMin : INT := 0;

    (* === ДДЮТ:НОВОЕ — счётчик промывок НФ (двухстадийный алгоритм,   *)
    (* см. блок 4а PRG_Fountain.st). RETAIN — переживает пропадание     *)
    (* питания, как и остальные счётчики/журналы в проекте.             *)
    iNfLastOnHour  : INT;   // время последнего включения НФ
    iNfLastOnMin   : INT;
    iNfLastOnDay   : INT;
    iNfLastOnMonth : INT;
    iNfLastOnYear  : INT;
    iNfFlushStage  : INT;   // 0=ждём часть 1, 1=часть 1 выполнена, ждём часть 2
    xNfFlushReady  : BOOL := TRUE;  // защита от многократного счёта подряд
    iNfFlushCount  : INT;   // счётчик завершённых промывок (обе части)
    iNfFlushHour   : INT;   // время последней завершённой промывки
    iNfFlushMin    : INT;
    iNfFlushDay    : INT;
    iNfFlushMonth  : INT;
    iNfFlushYear   : INT;

    iNfRunMinAccum    : INT;
    iNfRunSecAccum    : DINT;
    iNfHealthySecLeft : DINT;    // (устар., не исп.)
    iNfHealthyHoursLeft : INT;   // (устар., не исп.)
    iNfHealthyMinLeft   : INT;   // (устар., не исп.)
    xNfProven         : BOOL;    // (устар., не исп.)
    xNfWorkPrev       : BOOL;    // === ДДЮТ:РЕАКТИВИРОВАНО === детект фронта для счётчика промывок (было "не исп.")
    iNfContinuousRunHour : INT;
    iNfContinuousRunMin  : INT;
    iNfContinuousRunSec  : INT;

    (* === ДДЮТ:НОВОЕ — счётчик промывок НФ (двухстадийный алгоритм) === *)
    xNfFirstScanDone : BOOL;   // защита от ложного фронта на первом скане
    iNfJustEndedSec  : INT;    // длительность только что завершённого интервала работы НФ, сек

    (* ===== БЛОКИРОВКА ДОЗАЦИИ ПРИ РУЧНОЙ ФИЛЬТРАЦИИ ======== *)
    xZapretDozacii : BOOL := TRUE;

    (* ===== ЗАПРЕТ ДОБОРА ВОДЫ ФОНТАНА (с экрана) ========== *)
    (* === ДДЮТ:НОВОЕ === Единый селектор заслонки, тот же          *)
    (* паттерн (0/1/2), что у остальных узлов. Раскладка —          *)
    (* PRG_Fountain.st блок 2а: 0=Ручной → xDamperForceOpen:=TRUE    *)
    (* (открыто несмотря ни на что); 1=Выкл → xDamperForceClose:=    *)
    (* TRUE И xDamperZapretDobor:=TRUE (закрыта и запрет на новый     *)
    (* добор); 2=Авто → обе форс-переменные и запрет сняты, работает *)
    (* обычная автоматика по датчикам (гистерезис + попытки).        *)
    (* xDamperZapretDobor САМА теперь НЕ RETAIN (см. ниже, non-retain*)
    (* блок) — вычисляется из iDamperSelect, а не пишется напрямую. *)
    iDamperSelect : INT := 2;   // заслонка: 0=ручной,1=выкл,2=авто

    (* ===== СВЕТ ==================================== *)
    (* === ДДЮТ:ИЗМЕНЕНО (единый селектор, заменяет iLightMode) === *)
    (* Старое трёхрежимное iLightMode (0=ручной вкл/выкл через     *)
    (* xLightManualOn, 1=принудительно вкл, 2=по закату) упразднено*)
    (* — раскладывается в тот же паттерн (Enable, ManualForce),    *)
    (* что и у остальных узлов. "Ручной пуск" здесь = force-вкл    *)
    (* независимо от расписания (использует уже существующий      *)
    (* xLightForceOn), "Авто" = штатная работа по закату.          *)
    iLightSelect : INT  := 2;       // свет: 0=ручной,1=выкл,2=авто(закат)
    iSoundMode   : INT  := 2;       // FUTURE_SOUND
    xSoundEnable : BOOL := TRUE;    // FUTURE_SOUND

    (* ===== === ДДЮТ:ИЗМЕНЕНО (v2) — РАСЧЁТ ЗАКАТА (NOAA+рефракция) *)
    (* Координаты объекта ДДЮТ — ПОДТВЕРЖДЕНО (44.61581/33.52276). *)
    (* Формат — десятичные градусы (не град/мин/сек), как и была     *)
    (* организована переменная изначально — уточнять формат не       *)
    (* потребовалось, только сами значения.                          *)
    rSunLatitude          : REAL := 44.61581;  // широта объекта, град (-90..90)
    rSunLongitude         : REAL := 33.52276;  // долгота объекта, град (-180..180)
    (* === ДДЮТ:НОВОЕ === Запоминает долготу, на которую УЖЕ           *)
    (* среагировал автоподбор часового пояса (см. PRG_Fountain.st,     *)
    (* блок 11). По умолчанию совпадает с rSunLongitude — чтобы на     *)
    (* первом холодном старте НЕ переписать корректный дефолт          *)
    (* iChoseTimeZone=14 (+3, Москва) на неверный (см. пояснение там). *)
    rSunLongitudePrev     : REAL := 33.52276;
    (* === ДДЮТ:ИЗМЕНЕНО === часовой пояс теперь выбирается         *)
    (* КОМБОБОКСОМ через FB_TimeZoneSelect (индекс 0-23 → смещение  *)
    (* -11..+12). iChoseTimeZone — то, что крутит оператор на       *)
    (* экране ("Текстовый список", см. FB_TimeZoneSelect.st для     *)
    (* полного списка городов). 14 = Москва/Крым (+3) по умолчанию. *)
    (* === ДДЮТ:НОВОЕ === ТАКЖЕ теперь автоматически подбирается    *)
    (* ОДИН РАЗ при каждом реальном изменении долготы (не при        *)
    (* каждом цикле!) — см. PRG_Fountain.st блок 11. Если после      *)
    (* автоподбора оператор вручную поправит значение — это          *)
    (* сохранится и не будет затёрто повторно, пока долгота снова     *)
    (* не изменится.                                                  *)
    iChoseTimeZone        : INT  := 14;     // индекс часового пояса, с экрана (0..23)

    (* === ДДЮТ:ИЗМЕНЕНО (по макету экрана) === Коррекция теперь    *)
    (* ОДНО знаковое поле "+00мин"/"-00мин", а не два раздельных     *)
    (* элемента (было: минуты + отдельный тумблер раньше/позже).    *)
    (* Раскладывается на пару (iSunsetCorrectMin, xSunsetCorrectEarlier)*)
    (* — те, что реально идут на вход FB_SunsetRelay — в             *)
    (* PRG_Fountain.st блок 11, тем же приёмом, что и 3-позиционные  *)
    (* селекторы в блоке 2а.                                        *)
    iSunsetCorrectSigned  : INT  := 0;      // коррекция заката, мин, ЗНАКОВАЯ (- раньше, + позже)

    (* === ДДЮТ:ИЗМЕНЕНО === время отключения теперь РАЗДЕЛЬНО     *)
    (* для будних и выходных дней (было одно значение на все дни). *)
    iOffHourWeekday    : INT := 23;   // час отключения, будний день
    iOffMinuteWeekday  : INT := 0;    // минута отключения, будний день
    iOffHourWeekend    : INT := 23;   // час отключения, выходной день
    iOffMinuteWeekend  : INT := 0;    // минута отключения, выходной день

    (* === ДДЮТ:ИЗМЕНЕНО === FB_FountainSchedule — расписание         *)
    (* света и насосов реально управляет DO1/DO9 (в авто-режиме,      *)
    (* iLightSelect=2 / iPumpSelect=2 — см. PRG_Fountain.st блоки     *)
    (* 12/14). iLightScheduleMode/iPumpScheduleMode — ВНУТРЕННИЕ       *)
    (* переключатели самого расписания (не путать с внешними          *)
    (* iLightSelect/iPumpSelect!).                                     *)
    (* === ДДЮТ:ИЗМЕНЕНО (round 2) === Раньше у света и насосов было   *)
    (* по 4 ОДИНАКОВЫХ положения (полная симметрия). Теперь — РАЗНАЯ   *)
    (* кодировка, ВНИМАТЕЛЬНО:                                         *)
    (*   СВЕТ (4 положения):                                           *)
    (*     0 = Авто  — вкл. по фиксированному времени будни/выходные   *)
    (*         (iLightOnHourWeekday и т.д. ниже), выкл. — общий         *)
    (*         Off_Hour/Minute                                          *)
    (*     1 = Вкл   — горит постоянно, не выключается никогда          *)
    (*     2 = Выкл  — не включается никогда                            *)
    (*     3 = Астро — вкл. по расчёту заката (fbSunset), выкл. — тот   *)
    (*         же общий Off_Hour/Minute                                 *)
    (*   НАСОСЫ (3 положения — БЕЗ "Астро", убрали по факту, оказалось  *)
    (*   ненужным для насосов):                                         *)
    (*     0 = Авто  — вкл. по фиксированному времени (iPumpOnHourWeekday*)
    (*         и т.д.), выкл. — тот же общий Off_Hour/Minute            *)
    (*     1 = Вкл   — работает постоянно, не выключается никогда       *)
    (*     2 = Выкл  — не включается никогда                            *)
    (* В любом случае внешний селектор (iLightSelect/iPumpSelect)      *)
    (* должен быть = 2 ("Авто"), иначе эти переключатели ни на что     *)
    (* не влияют — см. блок 2а PRG_Fountain.st.                        *)
    (* ДЕФОЛТ СВЕТА = 3 (Астро) — сохраняем изначально задуманное      *)
    (* поведение "по умолчанию свет идёт по закату". ВАЖНО: это НЕ 0 — *)
    (* в новой кодировке 0 означает "Авто" (фиксированное время), это   *)
    (* другое поведение. Легко перепутать при переносе, если менять     *)
    (* кодировку не глядя на смысл дефолта.                             *)
    iLightScheduleMode : INT := 3;   // свет: 0=Авто,1=Вкл,2=Выкл,3=Астро (дефолт: по закату)
    iPumpScheduleMode  : INT := 0;   // насосы: 0=Авто,1=Вкл,2=Выкл (дефолт: по времени)

    iLightOnHourWeekday   : INT := 18;   // ручное расписание света: включение, будни
    iLightOnMinuteWeekday : INT := 0;
    iLightOnHourWeekend   : INT := 18;   // ручное расписание света: включение, выходные
    iLightOnMinuteWeekend : INT := 0;

    iPumpOnHourWeekday    : INT := 8;    // расписание насосов: включение, будни (база 8:00)
    iPumpOnMinuteWeekday  : INT := 0;
    iPumpOnHourWeekend    : INT := 8;    // расписание насосов: включение, выходные (база 8:00)
    iPumpOnMinuteWeekend  : INT := 0;

    (* === ДДЮТ:УДАЛИТЬ — заменены на пары Weekday/Weekend выше === *)
    (*
    iLightOffHour   : INT := 23;
    iLightOffMinute : INT := 0;
    *)

    (* ===== НАРАБОТКА В РУЧНОМ РЕЖИМЕ (RETAIN) ============== *)
    iNfManualRunMinBuffer : INT;
    iNfManualRunMinToday  : INT;
    iNfManualRunHourTotal : INT;
    iPhManualRunMinBuffer : INT;
    iAlgManualRunMinBuffer : INT;   // (устар., не исп.)
    iPhManualRunSecAccum : DINT;
    iPhManRunSec  : INT;
    iPhManRunHour : INT;
    iPhManRunMin  : INT;

    (* ===== НАКОПЛЕННАЯ НАРАБОТКА ДОЗАТОРОВ =============== *)
    iPhRunHourTotal : INT;
    iAlgRunHour : INT;
    iAlgRunMinBuffer2 : INT;
    iPhRunSecAccum : DINT;
    iPhRunSecDisp  : INT;
    iAlgRunSecAccum : DINT;
    iAlgRunSec  : INT;
    iPhStartCount  : INT;
    iAlgStartCount  : INT;

    (* ===== ДОЛГОВАЯ СИСТЕМА АЛЬГИЦИДА (RETAIN) ============= *)
    rAlgDebtSec         : REAL := 0.0;
    udiAlgLastDebtStamp : UDINT := 0;
    xAlgDebtInitDone    : BOOL := FALSE;
    iAlgLastDoseDay     : INT := 0;
    iAlgLastDoseMonth   : INT := 0;
    iAlgLastDoseYear    : INT := 0;
    iAlgLastDoseHourR   : INT := 0;
    iAlgLastDoseMinR    : INT := 0;
    iAlgLastDoseSecR    : INT := 0;

    (* ===== ДОЛГОВАЯ СИСТЕМА БИОПАГА (RETAIN) =============== *)
    rBioDebtSec         : REAL := 0.0;
    udiBioLastDebtStamp : UDINT := 0;
    xBioDebtInitDone    : BOOL := FALSE;
    iBioLastDoseDay     : INT := 0;
    iBioLastDoseMonth   : INT := 0;
    iBioLastDoseYear    : INT := 0;
    iBioLastDoseHourR   : INT := 0;
    iBioLastDoseMinR    : INT := 0;
    iBioLastDoseSecR    : INT := 0;
    iBioRunSecAccum     : DINT;
    iBioRunSecDisp      : INT;
    iBioStartCount      : INT;
    iBioManSetMin    : INT := 10;
    iBioManRemMinRaw    : INT;
    iBioManRemSecRaw    : INT;
END_VAR

VAR_GLOBAL
    (* === ДДЮТ:ИЗМЕНЕНО (round 3) === ЖУРНАЛ ИЗМЕНЕНИЙ ФОНТАНА: управление *)
    (* Свой экран пароля (не встроенный виджет OwenVisu), БЕЗ                *)
    (* промежуточного диалога "Вы уверены?" — сразу экран пароля.           *)
    (* Схема экрана (2 шага, было 3):                                       *)
    (*   1) Кнопка "Очистить журнал" → xAskClearFountainLog := TRUE          *)
    (*      (эта же переменная = видимость экрана пароля, второй             *)
    (*      переменной для промежуточного окна больше нет)                   *)
    (*   2) Экран пароля — поле ввода → iFountainLogPinEntry; кнопка          *)
    (*      "Войти"/"Подтвердить" → xFountainLogPinSubmit := TRUE;            *)
    (*      кнопка "Отмена" → xAskClearFountainLog := FALSE;                  *)
    (*      Всю проверку пароля и результат делает ST-код                    *)
    (*      (PRG_Fountain.st, блок 17а).                                      *)
    xAskClearFountainLog     : BOOL;   // = видимость экрана пароля (фонтан)
    iFountainLogPinEntry     : INT;    // ← сюда экран отдаёт введённое число
    xFountainLogPinSubmit    : BOOL;   // ← сюда экран отдаёт "нажали Войти"
    xFountainLogClearedMsg   : BOOL;   // TRUE на 3 сек — "Журнал сброшен"
    xFountainLogPassBadMsg   : BOOL;   // TRUE на 3 сек — "Пароль не подошёл"
    xFountainLogClear        : BOOL;   // реальный триггер очистки (пишет теперь ТОЛЬКО код, не экран)

    (* === ДДЮТ:ИЗМЕНЕНО (round 3) === Тот же набор для ЖУРНАЛА ПЧ           *)
    (* (GVL.sParamLog, GVL.xLogClear/xAskClearLog) — это твой скриншот.      *)
    (* Схема идентична фонтанному журналу выше (2 шага, без промежуточного   *)
    (* окна) — GVL.xAskClearLog сразу = видимость экрана пароля.             *)
    iPumpLogPinEntry     : INT;    // ← сюда экран отдаёт введённое число
    xPumpLogPinSubmit    : BOOL;   // ← сюда экран отдаёт "нажали Войти"
    xPumpLogClearedMsg   : BOOL;   // TRUE на 3 сек — "Журнал ПЧ сброшен"
    xPumpLogPassBadMsg   : BOOL;   // TRUE на 3 сек — "Пароль не подошёл"

    (* Защита от ложной записи "изменилось с 0 на дефолт" на самом первом *)
    (* скане после заливки/сброса — сначала просто СНИМАЕМ снимок текущих *)
    (* значений без сравнения, дальше сравниваем как обычно (тот же       *)
    (* приём, что и xLog_Initialized в журнале ПЧ, PRG_Pumps.st).         *)
    xFountainLogInitialized : BOOL;

    (* "Тени" (запомненное предыдущее значение) — по одной на каждый      *)
    (* отслеживаемый параметр. НЕ RETAIN — при перезапуске просто снова   *)
    (* делаем снимок (см. xFountainLogInitialized выше), это не потеря    *)
    (* данных, сам журнал (aFountainLog) отдельно и RETAIN.               *)
    iLogPrevFilterMinRunMin  : INT;
    iLogPrevUvNfMinRunMin    : INT;
    rLogPrevAlgDoseMlPerDay  : REAL;
    rLogPrevAlgFlowMlPerHour : REAL;
    rLogPrevBioDoseMlPerDay  : REAL;
    rLogPrevBioFlowMlPerHour : REAL;
    iLogPrevAlgManSetMin     : INT;
    iLogPrevBioManSetMin     : INT;
    iLogPrevPhSelect         : INT;
    iLogPrevAlgSelect        : INT;
    iLogPrevBioSelect        : INT;
    xLogPrevVseSist          : BOOL;
    (* === ДДЮТ:НОВОЕ (расширение списка) === *)
    iLogPrevDamperSelect     : INT;   // клапан добора, 3-поз (Ручной/Выкл/Авто)
    iLogPrevLightSelect      : INT;   // свет, 3-поз (внешний селектор)
    iLogPrevPumpSelect       : INT;   // насосы фонтана, 3-поз (внешний селектор)
    iLogPrevLevelSensorCount : INT;   // 2 или 3 датчика уровня
    iLogPrevLightScheduleMode : INT;  // расписание света, 0-3 (Авто/Вкл/Выкл/Астро)
    iLogPrevPumpScheduleMode  : INT;  // расписание насосов, 0-2 (Авто/Вкл/Выкл)
    iLogPrevLightOnHourWeekday   : INT;
    iLogPrevLightOnMinuteWeekday : INT;
    iLogPrevLightOnHourWeekend   : INT;
    iLogPrevLightOnMinuteWeekend : INT;
    iLogPrevPumpOnHourWeekday    : INT;
    iLogPrevPumpOnMinuteWeekday  : INT;
    iLogPrevPumpOnHourWeekend    : INT;
    iLogPrevPumpOnMinuteWeekend  : INT;
    iLogPrevOffHourWeekday       : INT;
    iLogPrevOffMinuteWeekday     : INT;
    iLogPrevOffHourWeekend       : INT;
    iLogPrevOffMinuteWeekend     : INT;
    iLogPrevSunsetCorrectSigned  : INT;
    iLogPrevChoseTimeZone        : INT;
    rLogPrevSunLatitude          : REAL;
    rLogPrevSunLongitude         : REAL;
    (* xAlarmReset и запуски таймерных доз — не "тени" значений, а       *)
    (* детект ФРОНТА момент-действия (RTRIG-style, вручную через Prev): *)
    xLogPrevAlarmReset       : BOOL;
    (* === ДДЮТ:НОВОЕ (второе расширение) === Гистерезисы уровня,      *)
    (* задержка выключения добора, уставки попыток добора — забыты в    *)
    (* первом списке, добавлены отдельно.                                *)
    iLogPrevLevel1DebounceSec   : INT;
    iLogPrevLevel2DebounceSec   : INT;
    iLogPrevLevel3DebounceSec   : INT;
    iLogPrevRefillOffDelayMin   : INT;
    iLogPrevRefillOffDelaySec   : INT;
    iLogPrevRefillDurHours      : INT;
    iLogPrevBetweenRefillHours  : INT;
    iLogPrevRefillAttemptsMax   : INT;

    (* === ДДЮТ:УДАЛИТЬ — УРОВЕНЬ В ЧАШЕ ПО АНАЛОГУ (AI1) ===== *)
    (*
    rWaterLevelRaw  : REAL;
    xMV110_8A_Error : BOOL;
    rWaterLevelCm   : REAL;
    xWaterSensorOk  : BOOL := TRUE;
    xLevelOverflow   : BOOL;
    xLevelAboveNorm  : BOOL;
    xLevelNeedRefill : BOOL;
    xLevelEmergency1 : BOOL;
    xLevelEmergency2 : BOOL;
    *)

    (* === ДДЮТ:ИЗМЕНЕНО (round 3) — УРОВЕНЬ ЧАШИ, 2 ИЛИ 3         *)
    (* ДИСКРЕТНЫХ ВХОДА (конфигурируется iLevelSensorCountPending) ===    *)
    (* Сухой ход больше НЕ отдельный физический вход (DI6 убран из *)
    (* карты) — он теперь ВЫЧИСЛЯЕТСЯ из Уровня1: если Уровень1=0   *)
    (* держится дольше гистерезиса — это и есть сухой ход.         *)
    xLevel1   : BOOL;   // ← DI7 Уровень1 (везде: 0=сухой ход)
    xLevel2   : BOOL;   // ← DI8 Уровень2 (везде: 0=старт добора; в режиме 2 датчиков ТАКЖЕ 1=стоп)
    xLevel3   : BOOL;   // ← DI12 Уровень3 (ТОЛЬКО режим 3 датчика: 1=стоп добора)

    xDryRunAlarm : BOOL;  // === ВЫЧИСЛЯЕТСЯ === Уровень1=0 подтверждено
                          // гистерезисом. НЕ защёлка — снимается
                          // автоматически когда Уровень1 вернулся в 1
                          // (держится гистерезис). Блокирует
                          // АВТОМАТИЧЕСКОЕ управление светом/насосами/
                          // добором/дозацией; ручное управление (форс-
                          // кнопки) работает отдельным условием через
                          // OR и дry-run НЕ перекрывает.

    (* === ДДЮТ:НОВОЕ === DI6 теперь — ОБРАТНАЯ СВЯЗЬ по DO13, а не  *)
    (* отдельный вход сухого хода. Сравниваем командуемое состояние  *)
    (* DO13 (= NOT xDryRunAlarm) с фактическим сигналом на DI6 —      *)
    (* расхождение дольше 10с считается аварией (тот же паттерн,     *)
    (* что и реле обратной связи дозаторов pH/альгицид/биопаг).      *)
    xDryRunRelayFb    : BOOL;   // ← DI6, факт подтверждения DO13
    xDryRunRelayAlarm : BOOL;   // авария: DO13 и DI6 разошлись >10с

    xLevel2LowConfirmed  : BOOL;  // Уровень2=0 подтверждено (старт добора)
    xLevel2HighConfirmed : BOOL;  // Уровень2=1 подтверждено (стоп, режим 2 датчика)
    xLevel3HighConfirmed : BOOL;  // Уровень3=1 подтверждено (стоп, режим 3 датчика)
    xRefillStartConfirmed : BOOL; // = xLevel2LowConfirmed (единая точка входа)
    xRefillEnoughConfirmed : BOOL; // = xLevel2HighConfirmed ИЛИ xLevel3HighConfirmed
                                   // (в зависимости от iLevelSensorCountPending)
    xRefillOffConfirmed : BOOL;   // xRefillEnoughConfirmed выдержан доп.
                                   // задержку iRefillOffDelayMin/Sec — реально закрываем

    (* === ДДЮТ: ОСТАВЛЕНО АКТИВНЫМ === На ДДЮТ ямы слива нет,   *)
    (* эти переменные нигде в PRG_Fountain не используются, но     *)
    (* нужны для компиляции PRG_PolivSPK.st (сохранён, не           *)
    (* вызывается). rSlivRaw всегда 0 (канал в дереве не привязан),*)
    (* PRG_PolivSPK физически не выполняется — влияния на работу    *)
    (* системы нет.                                                 *)
    rSlivRaw     : REAL;
    rSlivLevelCm : REAL;
    (* === ДДЮТ:УДАЛИТЬ === не используются нигде (были для полива *)
    (* травы, которого на ДДЮТ нет) *)
    (*
    xPolivEnable : BOOL;
    xDoborBochki : BOOL;
    *)

    (* ===== ЗАСЛОНКА (КЛАПАН ДОБОРА) — DO11 =============== *)
    xDamperCmdOpen    : BOOL;        // → DO11: 1=открыть (добор), 0=закрыть
    (* === ДДЮТ:НОВОЕ === Теперь ВЫЧИСЛЯЮТСЯ из iDamperSelect (см.    *)
    (* RETAIN-блок выше и PRG_Fountain.st блок 2а), не редактируются  *)
    (* напрямую с экрана. Работают НЕЗАВИСИМО от автоматики через OR  *)
    (* — даже при подтверждённом сухом ходе (xDryRunAlarm) "Ручной"    *)
    (* режим принудительно открывает клапан (автоматика при этом      *)
    (* всё равно остаётся заблокированной, пока сухой ход не снимется)*)
    xDamperForceOpen   : BOOL;       // = "Ручной" (iDamperSelect=0)
    xDamperForceClose  : BOOL;       // = "Выкл" (iDamperSelect=1)
    xDamperZapretDobor : BOOL;       // = "Выкл" (iDamperSelect=1), запрет нового добора
    (* Статус для экрана *)
    sDamperPosition   : WSTRING(20); // "Добор ВКЛ" / "Добор ВЫКЛ"
    sDamperFullStatus : WSTRING(50); // = sDamperPosition (упрощено, нет режима)

    (* === ДДЮТ:НОВОЕ — авария аварийного потолка добора === *)
    (* xRefillMaxDurationAlarm убрана — заменена xRefillAttemptsAlarm  *)
    (* (объявлена выше, в блоке возвращённой системы попыток).         *)

    (* === ДДЮТ:НОВОЕ === Готовая логическая переменная "у нас       *)
    (* только 2 датчика уровня" — вычисляется из iLevelSensorCountPending*)
    (* каждый цикл (PRG_Fountain.st, блок 2а). Используй её для      *)
    (* свойства "Невидимость" элементов Уровня3 на экране заслонки   *)
    (* (лампа Уровень3, гистерезис tLevel3DebounceSec и т.п.) —       *)
    (* когда TRUE, эти элементы прячь. Отдельной переменной "только  *)
    (* 3 датчика" не заводил — если понадобится, это просто           *)
    (* NOT xOnlyTwoLevels, привязывай к ней напрямую с отрицанием    *)
    (* в свойстве видимости, если у визуализации так удобнее.        *)
    xOnlyTwoLevels : BOOL;   // TRUE = iLevelSensorCountPending = 2 (датчика Уровень3 физически нет)

    (* === ДДЮТ:ВОЗВРАЩЕНО — система попыток добора === *)
    (* iRefillAttempts НЕ RETAIN — так было и в Саки (сбрасывается    *)
    (* при перезапуске контроллера, а не только вручную/по успеху).   *)
    iRefillAttempts   : INT;   // текущее число неудачных попыток подряд
    (* xRefillActivePrev — БОЛЬШЕ НЕ НУЖНА. Раньше вручную детектили   *)
    (* фронт начала новой попытки, чтобы принудительно сбросить        *)
    (* tonRefillTry. Упростили: стандартное поведение TON само         *)
    (* сбрасывает отсчёт в 0 при IN=FALSE и считает заново при          *)
    (* IN=TRUE — отдельный флаг для этого не требуется.                *)
    xRefillPauseRun   : BOOL;  // идёт пауза между неудачными попытками

    (* Авария: все попытки израсходованы, лимит превышен. Не путать  *)
    (* с xDryRunAlarm (тот про сам факт нехватки воды прямо сейчас,   *)
    (* этот — про то, что автоматика долго не может добиться "хватит"*)
    xRefillAttemptsAlarm : BOOL;

    (* === ДДЮТ:УДАЛИТЬ — концевики/реле направления заслонки === *)
    (* На ДДЮТ у заслонки нет концевиков DI13/DI14 и реле         *)
    (* направления DI15/DI16 — простой клапан по команде.         *)
    (*
    xDamperLimitOpen  : BOOL;
    xDamperLimitClose : BOOL;
    xDamperRelayOpen  : BOOL;
    xDamperRelayClose : BOOL;
    xDamperOpening    : BOOL;
    xDamperClosing    : BOOL;
    xDamperSensorFault : BOOL;
    xDamperAlarm      : BOOL;
    xDamperAutoMode   : BOOL;
    sDamperMode       : WSTRING(20);
    xLevelNormConfirmed   : BOOL;
    xLevelRefillConfirmed : BOOL;
    rRefillLevelStart : REAL;
    eDamperState      : E_DamperState;
    xDamperManualOpen  : BOOL;
    xDamperManualClose : BOOL;
    xDamperManualMode  : BOOL;
    *)

    (* ===== РАЗРЕШЕНИЯ И ФИЛЬТРАЦИЯ ======================= *)
    xPermissionToWork : BOOL;        // = xVseSist AND NOT xDryRunAlarm
    xNfWork           : BOOL;        // НФ работает СЕЙЧАС (по DI5)
    xNfHealthy        : BOOL;        // НФ исправен (непрерывная наработка)
    xNfPermission     : BOOL;
    xBlokDozacii      : BOOL;
    xFiltrationBlock  : BOOL;        // === ДДЮТ: всегда FALSE (нет аварийных уровней по см) ===

    (* === ДДЮТ:УДАЛИТЬ — двухуровневая блокировка по см ===== *)
    (*
    xAllSystemsBlock  : BOOL;
    xDO13DO14Block    : BOOL;
    xLeakAlarm        : BOOL;
    *)

    (* ========================================================= *)
    (* === ДДЮТ:УДАЛИТЬ — СВЯЗЬ С ПР200 (не используется, файл    *)
    (* PRG_PR200.st сохранён но не вызывается — вернуть легко)    *)
    (* ========================================================= *)
    (*
    xPr_ControlFromSpk : BOOL;
    wPr_Heartbeat      : WORD;
    iPr_SuhoyHod_Set   : INT := 5;
    iPr_Podpitka_Set   : INT := 60;
    iPr_Norma_Set      : INT := 80;
    iPr_Pereliv_Set    : INT := 90;
    iPr_DelaySec_Set   : INT := 60;
    xPr_PolivCmd       : BOOL;
    xPr_DoborCmd       : BOOL;
    xPr_ZapretPoliv    : BOOL;
    xPr_ZapretDobor    : BOOL;
    xPr_RuchnoyPoliv   : BOOL;
    xPr_RuchnoyDobor   : BOOL;
    xPr_RuchnoySliv    : BOOL;
    iPr_LevelCm        : INT;
    xPr_PolivActive    : BOOL;
    xPr_DoborActive    : BOOL;
    xPr_SlivActive     : BOOL;
    xPr_ErrDobor       : BOOL;
    xPr_ErrSliv        : BOOL;
    xPr_ErrPoliv       : BOOL;
    xPr_CommError      : BOOL;
    xPr_RawError       : BOOL;
    wPr_CmdWrite       : WORD;
    wPr_StatusRead     : WORD;
    sPr_Status         : WSTRING(40);
    *)

    (* ===== ВЫХОДЫ-КОМАНДЫ ================================ *)
    (* === ДДЮТ:УДАЛИТЬ — xUvCmd остаётся, но выхода нет === *)
    xUvCmd    : BOOL;                // считается для мониторинга/будущего, на DO НЕ подан
    xPumpsCmd : BOOL;                // → DO9
    xLightCmd : BOOL;                // → DO1

    (* ===== pH (только разрешение) ======================== *)
    (* === ДДЮТ:НОВОЕ === xPhEnable теперь ВЫЧИСЛЯЕТСЯ из          *)
    (* iPhSelect (см. PRG_Fountain.st блок 2а), не редактируется   *)
    (* напрямую с экрана.                                          *)
    xPhEnable    : BOOL;
    xPhRunCmd    : BOOL;
    xPhOutput    : BOOL;             // → DO16
    xPhRelayFb   : BOOL;             // ← DI9
    xPhManualRun : BOOL;
    iPhRunMinToday  : INT;
    iPhRunMinBuffer : INT;
    (* === ДДЮТ:НОВОЕ — авария реле обратной связи pH === *)
    xPhRelayAlarm : BOOL;            // команда есть, DI9 не подтвердил 10с

    (* ===== АЛЬГИЦИД (с таймером) =========================== *)
    (* === ДДЮТ:НОВОЕ === вычисляется из iAlgSelect === *)
    xAlgEnable    : BOOL;
    xAlgRunCmd    : BOOL;
    xAlgOutput    : BOOL;             // → DO14
    iAlgAutoStartCount : INT;
    xAlgRelayFb   : BOOL;             // ← DI11
    xAlgManualRun : BOOL;
    iAlgManRunSecAccum  : DINT;
    iAlgManRunHour : INT;
    iAlgManRunMin  : INT;
    iAlgManRunSec   : INT;
    xAlgManualTimeStart : BOOL;
    xAlgManualTimeStop  : BOOL;
    xAlgManualTimeRun   : BOOL;
    (* === ДДЮТ:НОВОЕ === Диалог подтверждения калибровочной дозы.    *)
    (* Кнопка "Старт" на экране теперь пишет СЮДА (не в                *)
    (* xAlgManualTimeStart напрямую) — показывает окно с текстом       *)
    (* "Внимание, Альгицид будет переведён в Режим Выкл, не забудьте   *)
    (* вернуть его в Автоматический режим после завершения             *)
    (* отладочных работ!!!". Кнопка "Подтвердить" на этом окне делает  *)
    (* ДВА действия разом: GVL_Fountain.iAlgSelect := 1; и             *)
    (* GVL_Fountain.xAlgManualTimeStart := TRUE; затем сама себя        *)
    (* гасит := FALSE. Кнопка "Отмена" просто := FALSE.                *)
    xAskAlgManualTimeStart : BOOL;
    iAlgManSetMin    : INT;
    iAlgManRemMinRaw    : INT;
    iAlgManRemSecRaw    : INT;
    iAlgManRemHour   : INT;
    iAlgManRemMin : INT;
    iAlgManRemSec : INT;
    rAlgRemainSec  : REAL;
    iAlgRemainHour : INT;
    iAlgRemainMin  : INT;
    iAlgRemainSec  : INT;
    rAlgNextDoseSec : REAL;
    iAlgNextHour : INT;
    iAlgNextMin  : INT;
    iAlgNextSec  : INT;
    rAlgDoseSecCalc : REAL;
    iAlgDoseHour : INT;
    iAlgDoseMin : INT;
    iAlgDoseSec : INT;
    iAlgRunMin  : INT;
    iAlgRunMinBuffer : INT;
    iAlgStartToday   : INT;
    xAlgAlarm        : BOOL;
    rAlgFlowLPerHour : REAL;
    xAlgDosing           : BOOL;
    sAlgDosingStatus     : WSTRING(10);
    iAlgDebtMin      : INT;
    iAlgDebtSec      : INT;
    iAlgDebtHour     : INT;
    sAlgLastDebtTime : WSTRING(30);
    iAlgLastDoseHour : INT;
    iAlgLastDoseMin  : INT;
    iAlgLastDoseSec  : INT;
    sAlgLastDoseTime : WSTRING(30);
    (* === ДДЮТ:НОВОЕ — авария реле обратной связи альгицида === *)
    xAlgRelayAlarm : BOOL;            // команда есть, DI11 не подтвердил 10с

    (* ===== БИОПАГ — все переменные (не RETAIN) ============= *)
    xBioRunCmd          : BOOL;
    xBioOutput          : BOOL;            // → DO15
    xBioRelayFb         : BOOL;            // ← DI10
    xBioDosing          : BOOL;
    sBioDosingStatus    : WSTRING(10);
    rBioDoseSecCalc     : REAL;
    iBioDoseHour    : INT;
    iBioDoseMin     : INT;
    iBioDoseSec     : INT;
    iBioDebtHour        : INT;
    iBioDebtMin         : INT;
    iBioDebtSec         : INT;
    rBioNextDoseSec     : REAL;
    iBioNextHour    : INT;
    iBioNextMin     : INT;
    iBioNextSec     : INT;
    iBioRunHour : INT;
    iBioRunMin  : INT;
    iBioRunSec   : INT;
    iBioStartToday      : INT;
    iBioDebtDays        : INT;
    iAlgDebtDays        : INT;
    sBioLastDebtTime    : WSTRING(30);
    sBioLastDoseTime    : WSTRING(30);
    iBioLastDoseHour    : INT;
    iBioLastDoseMin     : INT;
    iBioLastDoseSec     : INT;
    xBioAlarm           : BOOL;
    rBioFlowLPerHour    : REAL;
    tonBioDebtTick      : TON;
    tonBioRunTick       : TON;
    (* === ДДЮТ:НОВОЕ === вычисляется из iBioSelect === *)
    xBioEnable             : BOOL;
    xBioManualRun          : BOOL;
    iBioManRunSecAccum  : DINT;
    iBioManRunHour : INT;
    iBioManRunMin  : INT;
    iBioManRunSec   : INT;
    tonBioManualTick       : TON;
    xBioManualTimeStart : BOOL;
    xBioManualTimeStop  : BOOL;
    xBioManualTimeRun   : BOOL;
    (* === ДДЮТ:НОВОЕ === Тот же диалог, что и у альгицида (см. там), *)
    (* текст предупреждения аналогичный, но про Биопаг.                *)
    xAskBioManualTimeStart : BOOL;
    iBioManRemHour    : INT;
    iBioManRemMin : INT;
    iBioManRemSec : INT;
    tonBioManualSecTick  : TON;
    (* === ДДЮТ:НОВОЕ — авария реле обратной связи биопага === *)
    xBioRelayAlarm : BOOL;            // команда есть, DI10 не подтвердил 10с

    (* ===== СВЕТ ========================================== *)
    (* === ДДЮТ:УДАЛИТЬ — расписание по DI7 (теперь уровень) === *)
    (*
    xLightOnSchedule : BOOL;
    xLightRelayState : BOOL;
    *)
    (* === ДДЮТ:УДАЛИТЬ — заменена единым селектором iLightSelect *)
    (* Было: xLightManualOn : BOOL; — переменная убрана целиком.  *)
    (* === ДДЮТ:НОВОЕ === xLightEnable теперь ВЫЧИСЛЯЕТСЯ из       *)
    (* iLightSelect (см. PRG_Fountain.st блок 2а).                 *)
    xLightEnable     : BOOL;
    xLightForceOn    : BOOL;          // = "ручной пуск" (iLightSelect=0), OR-приоритет
    xLightFault      : BOOL;          // всегда FALSE (диагностика не актуальна)

    (* === ДДЮТ:ИЗМЕНЕНО (v2) — РАСЧЁТ ЗАКАТА (диагностика для экрана) === *)
    (* === ДДЮТ:НОВОЕ === результат FB_TimeZoneSelect (для показа и *)
    (* для передачи в fbSunset). НЕ RETAIN — пересчитывается каждый *)
    (* цикл из iChoseTimeZone.                                      *)
    rSunTimeZone       : REAL;   // вычисленное смещение UTC, знаковое (fbTimeZone.TimeZone)

    (* === ДДЮТ:ИЗМЕНЕНО === разложение знакового iSunsetCorrectSigned*)
    (* на пару, которую реально ждёт FB_SunsetRelay. НЕ RETAIN —      *)
    (* пересчитывается каждый цикл, см. PRG_Fountain.st блок 11.      *)
    iSunsetCorrectMin     : INT;    // = ABS(iSunsetCorrectSigned)
    xSunsetCorrectEarlier : BOOL;   // = (iSunsetCorrectSigned < 0)

    xSunsetActive      : BOOL;   // текущее состояние авто-расчёта (fbSunset.Sunset_Auto)
    xSunsetCoordError  : BOOL;   // ошибка координат (широта/долгота вне диапазона)
    iSunsetHourCalc    : INT;    // расчётный час заката
    iSunsetMinuteCalc  : INT;    // расчётная минута заката
    iSunsetTimeLeftH   : INT;    // осталось до смены состояния, часы
    iSunsetTimeLeftM   : INT;    // осталось до смены состояния, минуты
    iSunsetDayOfYear   : INT;    // порядковый день года (диагностика)
    xIsWeekend         : BOOL;   // TRUE = суббота/воскресенье (алгоритм Зеллера)
    sCurrentDateStr    : WSTRING(12);  // текущая дата "дд.мм.гггг" для экрана

    (* === ДДЮТ:ПОДКЛЮЧЕНО — ВЫХОДЫ FB_FountainSchedule === *)
    (* xScheduleLightOut/xSchedulePumpOut теперь РЕАЛЬНО управляют    *)
    (* DO1/DO9 (в авто-режиме, см. PRG_Fountain.st блоки 12/14) —      *)
    (* было "только справочно", подключено по подтверждению.          *)
    xScheduleLightOut      : BOOL;   // = fbSchedule.Light_Out, участвует в DO1
    xSchedulePumpOut       : BOOL;   // = fbSchedule.Pump_Out, участвует в DO9
    iScheduleLightOnHour   : INT;    // итоговое время вкл. света сегодня (справочно)
    iScheduleLightOnMinute : INT;
    iScheduleOffHour       : INT;    // итоговое время выкл. фонтана сегодня (справочно)
    iScheduleOffMinute     : INT;
    iSchedulePumpOnHour    : INT;    // итоговое время вкл. насосов сегодня (справочно)
    iSchedulePumpOnMinute  : INT;

    (* === ДДЮТ:НОВОЕ — флаги видимости элементов на экране "График *)
    (* Фонтана" (4-позиционный режим). Привязывай свойство            *)
    (* "Невидимость"/"Видимость" элементов ровно к этим переменным —  *)
    (* никаких выражений/сравнений прямо на экране писать не нужно.  *)
    xLightShowInputFields   : BOOL;  // Режим света=1(Авто) → показать поля ввода будни/выходные
    xLightShowComputedTime  : BOOL;  // Режим света=0 или 1 → показать итоговое время (не заглушку)
    xLightShowAlwaysOnText  : BOOL;  // Режим света=2(Вкл) → текст "Вкл ручн"
    xLightShowAlwaysOffText : BOOL;  // Режим света=3(Выкл) → текст "Выкл ручн"
    xPumpShowInputFields    : BOOL;  // Режим насосов=1(Авто) → показать поля ввода будни/выходные
    xPumpShowComputedTime   : BOOL;  // Режим насосов=0 или 1 → показать итоговое время
    xPumpShowAlwaysOnText   : BOOL;  // Режим насосов=2(Вкл) → текст "Вкл ручн"
    xPumpShowAlwaysOffText  : BOOL;  // Режим насосов=3(Выкл) → текст "Выкл ручн"
    xOffTimeVisible         : BOOL;  // TRUE если хоть один из двух (свет ИЛИ насосы)
                                      // сейчас работает по времени (режим 0/1) —
                                      // привязать сюда видимость ВСЕХ 6 полей времени
                                      // выключения (см. ЭКРАНЫ_ДДЮТ.txt)

    (* === ДДЮТ:НОВОЕ === Флаги "внешний селектор перебивает расписание" *)
    (* ⚠️ НЕ ПУТАТЬ с четырьмя выше — те про iLightScheduleMode/          *)
    (* iPumpScheduleMode (ВНУТРЕННИЙ режим 0-3: Астро/Авто/Вкл/Выкл).     *)
    (* Эти четыре — про ДРУГУЮ, ВНЕШНЮЮ пару iLightSelect/iPumpSelect     *)
    (* (0=Ручной,1=Выкл,2=Авто, экран "Свет/Насосы"). Если внешний        *)
    (* селектор НЕ на "Авто" (=2) — итоговое время из FB_FountainSchedule *)
    (* просто НЕ ДЕЙСТВУЕТ на DO1/DO9, хотя продолжает считаться и        *)
    (* отображаться, как будто оно актуально. Эти флаги — предупреждение  *)
    (* оператору, что расписание сейчас не при делах. Вычисляются в       *)
    (* блоке 2а PRG_Fountain.st, ПРЯМО как готовые булевы (не выражения    *)
    (* на экране — история с опечаткой "FASLE" научила).                  *)
    xLightOuterForcedOn  : BOOL;  // iLightSelect=0(Ручной) — свет ВСЕГДА вкл, расписание не участвует
    xLightOuterForcedOff : BOOL;  // iLightSelect=1(Выкл)   — свет ВСЕГДА выкл, расписание не участвует
    xPumpOuterForcedOn   : BOOL;  // iPumpSelect=0(Ручной)  — насосы ВСЕГДА вкл, расписание не участвует
    xPumpOuterForcedOff  : BOOL;  // iPumpSelect=1(Выкл)    — насосы ВСЕГДА выкл, расписание не участвует

    (* ===== НАСОСЫ ФОНТАНА (ручное) ======================= *)
    (* === ДДЮТ:НОВОЕ === xManualPermissionNasos теперь          *)
    (* ВЫЧИСЛЯЕТСЯ из iPumpSelect (см. PRG_Fountain.st блок 2а).  *)
    xManualPermissionNasos : BOOL;
    xPumpsManualOn : BOOL;           // (устар.)
    xPumpsForceOn  : BOOL;           // = "ручной пуск" (iPumpSelect=0), OR-приоритет

    (* ===== ЗВУК (FUTURE_SOUND) =========================== *)
    xSoundOnSchedule : BOOL;
    xSoundOutput     : BOOL;
    xSoundManualOn   : BOOL;

    (* ===== ФИЛЬТРАЦИЯ (мониторинг) ======================= *)
    (* === ДДЮТ:ИЗМЕНЕНО — новая карта DI, см. PRG_Fountain блок 2 *)
    xFilter1Drive     : BOOL;        // ← DI1 (ПЧ1 насос фонтана)
    xFilter2Drive     : BOOL;        // ← DI2 (ПЧ2 насос фонтана)
    xDriveStart       : BOOL;        // ← DI3 (разрешение частотников)
    xUvContactor      : BOOL;        // ← DI4 (контактор УФ)
    xFilter1Contactor : BOOL;        // ← DI5 (контактор фильтр.насоса, для наработки НФ)
    xManualFilter     : BOOL;        // ручное вкл фильтрации с экрана
    (* === ДДЮТ:УДАЛИТЬ — не используются на ДДЮТ === *)
    (*
    xFilter2Contactor : BOOL;
    xFilter3Contactor : BOOL;
    xBarrelStart      : BOOL;
    *)

    (* ===== АВАРИИ ======================================== *)
    (* === ДДЮТ:УДАЛИТЬ — аварии несуществующего оборудования === *)
    (*
    xAlarmOverflow      : BOOL;
    xAlarmWaterSensor   : BOOL;
    *)
    (* === ДДЮТ:УДАЛИТЬ — старая авария "исчерпаны попытки" под       *)
    (* именем из Саки. Возвращена под новым именем                    *)
    (* xRefillAttemptsAlarm (объявлена выше, в блоке системы попыток).*)
    (* xAlarmRefillTimeout : BOOL; *)
    xAlarmFountain      : BOOL;      // → DO2 (мигает)
    xAlarmReset         : BOOL;

    (* ===== ФЛАГИ ПОДТВЕРЖДЕНИЯ СБРОСА ==================== *)
    xAskResetPh     : BOOL := FALSE;
    xAskResetAlg    : BOOL := FALSE;
    xAskResetBio    : BOOL := FALSE;
    xAskResetRefill : BOOL := FALSE;
    xAskResetNfFlush : BOOL := FALSE;  // === ДДЮТ:НОВОЕ === диалог "Сбросить счётчик промывок?"
    xAskResetAll    : BOOL := FALSE;
    xAskResetAlarms : BOOL := FALSE;
    xConfirmResetPh  : BOOL := FALSE;
    xConfirmResetAlg : BOOL := FALSE;
    xConfirmResetBio : BOOL := FALSE;
    xConfirmResetAll : BOOL := FALSE;
    (* === ДДЮТ:НОВОЕ === Раньше сброс попыток добора и промывок НФ был *)
    (* ЦЕЛИКОМ на стороне кнопки визуализации (без ST-кода вообще —      *)
    (* см. комментарии у xAskResetRefill/xAskResetNfFlush в коде          *)
    (* PRG_Fountain.st). Для журнала изменений это не годится — если      *)
    (* ST-код ни разу не выполняется, логировать нечего. Добавлены        *)
    (* обычные confirm-флаги, как у pH/альгицид/биопаг выше — кнопка      *)
    (* "Подтвердить" теперь пишет СЮДА (одно присвоение вместо трёх),     *)
    (* остальное (сам сброс + запись в журнал) делает ST-код.             *)
    xConfirmResetRefill  : BOOL := FALSE;
    xConfirmResetNfFlush : BOOL := FALSE;

    (* ===== МИГАНИЕ ====================================== *)
    xBlinkFast : BOOL;
    xBlinkSlow : BOOL;

    (* ===== СТРОКОВЫЕ СТАТУСЫ ============================= *)
    sVseSistStatus    : WSTRING(30);
    sPermissionStatus : WSTRING(30);
    sNfEnableStatus   : WSTRING(30);
    sPhStatus         : WSTRING(30);
    sAlgStatus         : WSTRING(30);
    sBioStatus         : WSTRING(30);
    sLightStatus      : WSTRING(30);
    sSoundStatus      : WSTRING(30);
    sRefillStatus     : WSTRING(30);
    sAlarmStopStatus  : WSTRING(30);
    sAlarmCauses      : WSTRING(255);
    sNfStatus         : WSTRING(30);
    sNfHealthyStatus  : WSTRING(30);
    (* === ДДЮТ:УДАЛИТЬ — статусы несуществующего === *)
    (*
    sDamperStatus     : WSTRING(30);
    sOverflowStatus   : WSTRING(30);
    sPolivStatus      : WSTRING(30);
    sLightFaultStatus : WSTRING(30);
    *)

    (* ===== ВРЕМЯ (RTC) ================================== *)
    iCurrentYear         : INT;
    iCurrentMonth        : INT;
    iCurrentDay          : INT;
    iCurrentHour         : INT;
    iCurrentMinute       : INT;
    iCurrentSecond       : INT;
    iCurrentTotalMinutes : INT;

    (* ========================================================= *)
    (* === ДДЮТ:УДАЛИТЬ — СВЯЗЬ С ПР200 (полив/слив) ============ *)
    (* Файл PRG_PR200.st сохранён, но не вызывается. Легко        *)
    (* вернуть — раскомментировать вызов в PLC_PRG и поднять       *)
    (* канал в дереве. Пока не удаляем эти переменные физически,  *)
    (* т.к. на них ссылается PRG_PR200.st, который держим          *)
    (* компилируемым.                                              *)
    (* ========================================================= *)
wPr200SuhoyHod_Net  : WORD;
wPr200Podpitka_Net  : WORD;
wPr200Norma_Net     : WORD;
wPr200Pereliv_Net   : WORD;
wPr200Delay_Net     : WORD;
wPr200LevelRead     : WORD;
wPr200StatusRead    : WORD;
rPr200SuhoyHod_Cur  : REAL;
rPr200Podpitka_Cur  : REAL;
rPr200Norma_Cur     : REAL;
rPr200Pereliv_Cur   : REAL;
rPr200Delay_Cur     : UDINT;
rPr200LevelCm       : REAL;
rPr200SuhoyHod_New  : REAL := 5.0;
rPr200Podpitka_New  : REAL := 60.0;
rPr200Norma_New     : REAL := 80.0;
rPr200Pereliv_New   : REAL := 90.0;
rPr200Delay_New     : UDINT := 60;
wPr200SuhoyHod_Write : WORD := REAL_TO_WORD(5);
wPr200Podpitka_Write : WORD := 60;
wPr200Norma_Write    : WORD := 80;
wPr200Pereliv_Write  : WORD := 90;
wPr200Delay_Write    : WORD := 60;
wPr200ApplyCmd       : WORD;
xPr200Online        : BOOL;
xPr200DoborActive   : BOOL;
xPr200SlivActive    : BOOL;
xPr200PolivActive   : BOOL;
xPr200ErrDobor      : BOOL;
xPr200ErrSliv       : BOOL;
xPr200ErrPoliv      : BOOL;
xApplyBtn           : BOOL;

    (* ========================================================= *)
    (* === ДДЮТ:УДАЛИТЬ — РЕЗЕРВНАЯ ЛОГИКА ПОЛИВА НА СПК ========= *)
    (* Файл PRG_PolivSPK.st сохранён, но не вызывается. На ДДЮТ   *)
    (* нет ямы слива — резерв полива физически не нужен. Оставлены*)
    (* декларации, т.к. на них ссылается PRG_PolivSPK.st.         *)
    (* ========================================================= *)
xSpkPolivMode    : BOOL;
xSpkRawDI17 : BOOL;
xSpkRawDI18 : BOOL;
xSpkPolivMode_OLD : BOOL;
xPr200OnlineStable : BOOL;
iPr200CommFilterSec : INT := 3;
xSpkLevelSensorOk : BOOL;
xMsgPr200Offline : BOOL := FALSE;
xMsgSpkNoSensor  : BOOL := FALSE;
xSpkDI_Dobor     : BOOL;
xSpkDI_Poliv     : BOOL;
xSpkDO_Dobor     : BOOL;
xSpkDO_Poliv     : BOOL;
xSpkRuchDobor    : BOOL;
xSpkRuchPoliv    : BOOL;
xSpkZapDobor     : BOOL;
xSpkZapPoliv     : BOOL;
xSpkDoborOn      : BOOL;
xSpkPolivOn      : BOOL;
xSpkErrDobor     : BOOL;
xSpkErrPoliv     : BOOL;
xSpkErrPereliv   : BOOL;
iSpkErrDelaySec  : INT := 5;
sSpkDoborStatus  : WSTRING(20);
sSpkPolivStatus  : WSTRING(20);
sSpkManualStatus : WSTRING(30);
wSpkMV_Inputs   : WORD;
xSpkMV_Error    : BOOL;
xSpkDI          : ARRAY[1..16] OF BOOL;
wSpkMU_Outputs     : WORD := 0;
wSpkMU_OutputsRead : WORD;
xSpkMU_Error       : BOOL;
wSpkMU_SafeOutputs : WORD := 0;
xSpkMU_WriteSafe   : BOOL := FALSE;
xSpkDO             : ARRAY[1..16] OF BOOL := [16(FALSE)];
rSpkLevelRaw    : REAL;
xSpkAI_Error    : BOOL;
END_VAR

(* ---- F_FaultCodeToText.st ---- *)
FUNCTION F_FaultCodeToText : WSTRING(100)
(* === ДДЮТ: без изменений относительно Саки Пруд === *)
VAR_INPUT
    eType    : E_PumpType;
    wCode    : WORD;
END_VAR
VAR
    wCleanCode : WORD;
    iCode      : INT;
END_VAR

CASE eType OF

    E_PumpType.PUMP:
        wCleanCode := wCode AND 16#7FFF;
        iCode := WORD_TO_INT(wCleanCode);

        CASE iCode OF
            0:  F_FaultCodeToText := "Нет ошибок";
            1:  F_FaultCodeToText := "OC0: Перегруз по току в режиме Стоп";
            2:  F_FaultCodeToText := "OC1: Перегруз по току при ускорении";
            3:  F_FaultCodeToText := "OC2: Перегруз по току при замедлении";
            4:  F_FaultCodeToText := "OC3: Перегруз по току в работе";
            5:  F_FaultCodeToText := "OU1: Перенапряжение при ускорении";
            6:  F_FaultCodeToText := "OU2: Перенапряжение при замедлении";
            7:  F_FaultCodeToText := "OU3: Перенапряжение в работе";
            9:  F_FaultCodeToText := "LU: Низкое напряжение питания";
            10: F_FaultCodeToText := "OL2: Перегрузка ПЧ";
            11: F_FaultCodeToText := "OL1: Перегрузка двигателя по току";
            14: F_FaultCodeToText := "OH: Перегрев ПЧ";
            15: F_FaultCodeToText := "EF: Аварийная остановка";
            16: F_FaultCodeToText := "CO: Ошибка коммуникации Modbus";
            20: F_FaultCodeToText := "Обрыв сигнала ОС ПИД";
            24: F_FaultCodeToText := "LP: Нижний уровень аварии ОС ПИД";
            27: F_FaultCodeToText := "HP: Верхний уровень аварии ОС ПИД";
            28: F_FaultCodeToText := "LL: Сухой ход";
            29: F_FaultCodeToText := "tE: Превышено время работы";
            31: F_FaultCodeToText := "Pr: Ошибка записи параметра";
        ELSE
            CASE iCode OF
                64: F_FaultCodeToText := "UC0: Внутр. ошибка в Стоп";
                65: F_FaultCodeToText := "UC1: Внутр. ошибка при ускорении";
                66: F_FaultCodeToText := "UC2: Внутр. ошибка при замедлении";
                67: F_FaultCodeToText := "UC3: Внутр. ошибка в работе";
                68: F_FaultCodeToText := "OC0: Перегруз по току в Стоп";
                69: F_FaultCodeToText := "OC1: Перегруз по току при ускорении";
                70: F_FaultCodeToText := "OC2: Перегруз по току при замедлении";
                71: F_FaultCodeToText := "OC3: Перегруз по току в работе";
                80: F_FaultCodeToText := "OU0: Перенапряжение в Стоп";
                81: F_FaultCodeToText := "OU1: Перенапряжение при ускорении";
                82: F_FaultCodeToText := "OU2: Перенапряжение при замедлении";
                83: F_FaultCodeToText := "OU3: Перенапряжение в работе";
                88: F_FaultCodeToText := "LU0: Низкое напряжение в Стоп";
                89: F_FaultCodeToText := "LU1: Низкое напряжение при ускорении";
                90: F_FaultCodeToText := "LU2: Низкое напряжение при замедлении";
                91: F_FaultCodeToText := "LU3: Низкое напряжение в работе";
                92: F_FaultCodeToText := "OL0: Перегрузка ПЧ в Стоп";
                93: F_FaultCodeToText := "OL1: Перегрузка ПЧ при ускорении";
                94: F_FaultCodeToText := "OL2: Перегрузка ПЧ при замедлении";
                95: F_FaultCodeToText := "OL3: Перегрузка ПЧ в работе";
                96: F_FaultCodeToText := "OT0: Перегрузка двиг. в Стоп";
                97: F_FaultCodeToText := "OT1: Перегрузка двиг. при ускорении";
                98: F_FaultCodeToText := "OT2: Перегрузка двиг. при замедлении";
                99: F_FaultCodeToText := "OT3: Перегрузка двиг. в работе";
                100: F_FaultCodeToText := "OH0: Перегрев ПЧ в Стоп";
                101: F_FaultCodeToText := "OH1: Перегрев ПЧ при ускорении";
                102: F_FaultCodeToText := "OH2: Перегрев ПЧ при замедлении";
                103: F_FaultCodeToText := "OH3: Перегрев ПЧ в работе";
                104: F_FaultCodeToText := "ES: Авар. остановка / обрыв фазы";
            ELSE
                F_FaultCodeToText := WCONCAT("Ошибка PUMP код ", INT_TO_WSTRING(iCode));
            END_CASE;
        END_CASE;

    E_PumpType.MINI:
        iCode := WORD_TO_INT(wCode);
        IF (iCode <= 63) OR ((iCode >= 88) AND (iCode <= 91)) THEN
            F_FaultCodeToText := "Нет ошибок";
        ELSE
            CASE iCode OF
                64: F_FaultCodeToText := "UC0: Внутр. ошибка в Стоп";
                65: F_FaultCodeToText := "UC1: Внутр. ошибка при ускорении";
                66: F_FaultCodeToText := "UC2: Внутр. ошибка при замедлении";
                67: F_FaultCodeToText := "UC3: Внутр. ошибка в работе";
                68: F_FaultCodeToText := "OC0: Перегруз по току в Стоп";
                69: F_FaultCodeToText := "OC1: Перегруз по току при ускорении";
                70: F_FaultCodeToText := "OC2: Перегруз по току при замедлении";
                71: F_FaultCodeToText := "OC3: Перегруз по току в работе";
                80: F_FaultCodeToText := "OU0: Перенапряжение в Стоп";
                81: F_FaultCodeToText := "OU1: Перенапряжение при ускорении";
                82: F_FaultCodeToText := "OU2: Перенапряжение при замедлении";
                83: F_FaultCodeToText := "OU3: Перенапряжение в работе";
                92: F_FaultCodeToText := "OL0: Перегрузка ПЧ в Стоп";
                93: F_FaultCodeToText := "OL1: Перегрузка ПЧ при ускорении";
                94: F_FaultCodeToText := "OL2: Перегрузка ПЧ при замедлении";
                95: F_FaultCodeToText := "OL3: Перегрузка ПЧ в работе";
                96: F_FaultCodeToText := "OT0: Перегрузка двиг. в Стоп";
                97: F_FaultCodeToText := "OT1: Перегрузка двиг. при ускорении";
                98: F_FaultCodeToText := "OT2: Перегрузка двиг. при замедлении";
                99: F_FaultCodeToText := "OT3: Перегрузка двиг. в работе";
                100: F_FaultCodeToText := "OH0: Перегрев ПЧ в Стоп";
                101: F_FaultCodeToText := "OH1: Перегрев ПЧ при ускорении";
                102: F_FaultCodeToText := "OH2: Перегрев ПЧ при замедлении";
                103: F_FaultCodeToText := "OH3: Перегрев ПЧ в работе";
                104: F_FaultCodeToText := "ES: Авар. остановка / обрыв фазы";
            ELSE
                F_FaultCodeToText := WCONCAT("Ошибка MINI код ", INT_TO_WSTRING(iCode));
            END_CASE;
        END_IF;

END_CASE;

(* ---- F_FormatLogDateOnly.st ---- *)
FUNCTION F_FormatLogDateOnly : WSTRING(10)
(* === ДДЮТ:НОВОЕ === Дата в формате ДД.ММ.ГГГГ, БЕЗ времени — для     *)
(* сжатого журнала изменений параметров фонтана (F_FountainLogWrite).  *)
(* Не трогает существующую F_FormatLogTimestamp() (дата+время) —       *)
(* та используется журналом ПЧ и другими местами без изменений.        *)
VAR
    sDay   : WSTRING(4);
    sMonth : WSTRING(4);
END_VAR

IF GVL_Fountain.iCurrentDay < 10 THEN
    sDay := WCONCAT("0", INT_TO_WSTRING(GVL_Fountain.iCurrentDay));
ELSE
    sDay := INT_TO_WSTRING(GVL_Fountain.iCurrentDay);
END_IF;

IF GVL_Fountain.iCurrentMonth < 10 THEN
    sMonth := WCONCAT("0", INT_TO_WSTRING(GVL_Fountain.iCurrentMonth));
ELSE
    sMonth := INT_TO_WSTRING(GVL_Fountain.iCurrentMonth);
END_IF;

F_FormatLogDateOnly := WCONCAT(sDay, WCONCAT(".", WCONCAT(sMonth,
    WCONCAT(".", INT_TO_WSTRING(GVL_Fountain.iCurrentYear)))));

(* ---- F_FormatLogTimestamp.st ---- *)
FUNCTION F_FormatLogTimestamp : WSTRING(20)
(* === ДДЮТ: без изменений относительно Саки Пруд === *)
VAR
    sDay, sMon, sYear, sHour, sMin, sSec : WSTRING(4);
END_VAR
IF iCurrentDay < 10 THEN
    sDay := WCONCAT("0", INT_TO_WSTRING(iCurrentDay));
ELSE sDay := INT_TO_WSTRING(iCurrentDay); END_IF;
IF iCurrentMonth < 10 THEN
    sMon := WCONCAT("0", INT_TO_WSTRING(iCurrentMonth));
ELSE sMon := INT_TO_WSTRING(iCurrentMonth); END_IF;
sYear := INT_TO_WSTRING(iCurrentYear MOD 100);
IF (iCurrentYear MOD 100) < 10 THEN
    sYear := WCONCAT("0", sYear);
END_IF;
IF iCurrentHour < 10 THEN
    sHour := WCONCAT("0", INT_TO_WSTRING(iCurrentHour));
ELSE sHour := INT_TO_WSTRING(iCurrentHour); END_IF;
IF iCurrentMinute < 10 THEN
    sMin := WCONCAT("0", INT_TO_WSTRING(iCurrentMinute));
ELSE sMin := INT_TO_WSTRING(iCurrentMinute); END_IF;
IF iCurrentSecond < 10 THEN
    sSec := WCONCAT("0", INT_TO_WSTRING(iCurrentSecond));
ELSE sSec := INT_TO_WSTRING(iCurrentSecond); END_IF;
F_FormatLogTimestamp := WCONCAT(sDay, WCONCAT(".",
    WCONCAT(sMon, WCONCAT(".",
    WCONCAT(sYear, WCONCAT(" ",
    WCONCAT(sHour, WCONCAT(":",
    WCONCAT(sMin, WCONCAT(":", sSec))))))))));

(* ---- F_FountainLogWrite.st ---- *)
FUNCTION F_FountainLogWrite : BOOL
(* === ДДЮТ:ИЗМЕНЕНО (round 7, ФИНАЛЬНАЯ СХЕМА) === Позиция 1 — ВСЕГДА     *)
(* самая последняя запись. При новой записи всё содержимое сдвигается на   *)
(* 1 позицию вниз (сдвиг ОБЯЗАТЕЛЬНО с конца массива к началу — иначе       *)
(* затрёшь данные раньше, чем скопируешь), новая запись садится на 1.       *)
(* Когда достигнут предел (60) — самая старая запись (позиция 60) просто    *)
(* выпадает при сдвиге. Экран теперь может использовать ФИКСИРОВАННЫЕ       *)
(* индексы (aFountainLog[1], [2], [3]...) — никаких вычисляемых индексов,   *)
(* никакого риска выйти за границы массива.                                 *)
VAR_INPUT
    sChangeText : WSTRING(60);   (* полное понятное название параметра: старое→новое *)
END_VAR
VAR
    i : INT;
END_VAR

FOR i := 60 TO 2 BY -1 DO
    GVL_Fountain.aFountainLog[i] := GVL_Fountain.aFountainLog[i-1];
END_FOR;

GVL_Fountain.aFountainLog[1] := WCONCAT(F_FormatLogDateOnly(), WCONCAT(" ", sChangeText));

IF GVL_Fountain.iFountainLogCount < 60 THEN
    GVL_Fountain.iFountainLogCount := GVL_Fountain.iFountainLogCount + 1;
END_IF;

F_FountainLogWrite := TRUE;

(* ---- F_LightScheduleModeText.st ---- *)
FUNCTION F_LightScheduleModeText : WSTRING(12)
(* === ДДЮТ:НОВОЕ === Переводит iLightScheduleMode (0-3) в текст для    *)
(* журнала. ВНИМАНИЕ: кодировка ДРУГАЯ, чем у F_SelectModeText          *)
(* (тройные селекторы pH/альгицид/биопаг/свет/насосы/заслонка) — не      *)
(* перепутать! Здесь 0=Авто, а не Ручной.                                *)
VAR_INPUT
    iMode : INT;
END_VAR

CASE iMode OF
    0: F_LightScheduleModeText := "Авто";
    1: F_LightScheduleModeText := "Вкл";
    2: F_LightScheduleModeText := "Выкл";
    3: F_LightScheduleModeText := "Астро";
ELSE
    F_LightScheduleModeText := "?";
END_CASE;

(* ---- F_PumpLogWrite.st ---- *)
FUNCTION F_PumpLogWrite : BOOL
(* === ДДЮТ:ИЗМЕНЕНО (round 7, ФИНАЛЬНАЯ СХЕМА) === Та же схема сдвига,    *)
(* что у F_FountainLogWrite (см. подробный комментарий там) — позиция 1     *)
(* всегда самая свежая запись, сдвиг ОБЯЗАТЕЛЬНО с конца массива к началу.  *)
VAR_INPUT
    sChangeText : WSTRING(65);   (* готовая строка одной записи *)
END_VAR
VAR
    i : INT;
END_VAR

FOR i := 30 TO 2 BY -1 DO
    GVL.aPumpLog[i] := GVL.aPumpLog[i-1];
END_FOR;

GVL.aPumpLog[1] := sChangeText;

IF GVL.iPumpLogCount < 30 THEN
    GVL.iPumpLogCount := GVL.iPumpLogCount + 1;
END_IF;

F_PumpLogWrite := TRUE;

(* ---- F_PumpScheduleModeText.st ---- *)
FUNCTION F_PumpScheduleModeText : WSTRING(12)
(* === ДДЮТ:НОВОЕ === Переводит iPumpScheduleMode (0-2, БЕЗ "Астро") в  *)
(* текст для журнала. Своя, третья кодировка — не путать ни с            *)
(* F_SelectModeText, ни с F_LightScheduleModeText (у насосов режимов      *)
(* на один меньше, и нет положения "Астро" вообще).                       *)
VAR_INPUT
    iMode : INT;
END_VAR

CASE iMode OF
    0: F_PumpScheduleModeText := "Авто";
    1: F_PumpScheduleModeText := "Вкл";
    2: F_PumpScheduleModeText := "Выкл";
ELSE
    F_PumpScheduleModeText := "?";
END_CASE;

(* ---- F_SelectModeText.st ---- *)
FUNCTION F_SelectModeText : WSTRING(12)
(* === ДДЮТ:НОВОЕ === Переводит 0/1/2 (единый селектор pH/альгицид/     *)
(* биопаг/свет/насосы/заслонка) в читаемый текст для журнала изменений. *)
VAR_INPUT
    iMode : INT;
END_VAR

CASE iMode OF
    0: F_SelectModeText := "Ручной";
    1: F_SelectModeText := "Выкл";
    2: F_SelectModeText := "Авто";
ELSE
    F_SelectModeText := "?";
END_CASE;
